C03662=1146.416,331.049,-77.493,-176.659,8.929,148.817
C03663=1146.420,330.801,-77.460,-176.662,8.926,148.817
C03664=1146.424,330.554,-77.428,-176.665,8.922,148.817
C03665=1146.427,330.305,-77.394,-176.667,8.919,148.817
C03666=1146.431,330.057,-77.361,-176.670,8.914,148.816
C03667=1146.436,329.809,-77.329,-176.672,8.911,148.816
C03668=1146.440,329.561,-77.296,-176.675,8.907,148.816
C03669=1146.444,329.314,-77.262,-176.677,8.904,148.816
C03670=1146.448,329.066,-77.229,-176.680,8.900,148.815
C03671=1146.452,328.818,-77.196,-176.682,8.896,148.815
C03672=1146.456,328.571,-77.163,-176.685,8.892,148.815
C03673=1146.460,328.323,-77.130,-176.687,8.889,148.815
C03674=1146.464,328.075,-77.098,-176.690,8.886,148.814
C03675=1146.468,327.827,-77.065,-176.693,8.881,148.814
C03676=1146.472,327.579,-77.032,-176.695,8.878,148.814
C03677=1146.477,327.331,-76.998,-176.698,8.874,148.814
C03678=1146.480,327.083,-76.967,-176.700,8.871,148.814
C03679=1146.484,326.836,-76.933,-176.703,8.867,148.813
C03680=1146.489,326.589,-76.901,-176.705,8.863,148.813
C03681=1146.494,326.340,-76.868,-176.708,8.859,148.813
C03682=1146.497,326.093,-76.836,-176.711,8.856,148.813
C03683=1146.501,325.845,-76.802,-176.713,8.853,148.813
C03684=1146.506,325.597,-76.770,-176.716,8.849,148.812
C03685=1146.509,325.349,-76.737,-176.718,8.846,148.812
C03686=1146.513,325.102,-76.704,-176.721,8.841,148.812
C03687=1146.518,324.853,-76.672,-176.724,8.838,148.812
C03688=1146.522,324.606,-76.639,-176.726,8.834,148.811
C03689=1146.525,324.357,-76.607,-176.729,8.831,148.811
C03690=1146.530,324.110,-76.574,-176.731,8.828,148.811
C03691=1146.534,323.862,-76.541,-176.734,8.823,148.811
C03692=1146.537,323.614,-76.509,-176.736,8.820,148.811
C03693=1146.542,323.366,-76.476,-176.739,8.816,148.810
C03694=1146.546,323.119,-76.444,-176.742,8.813,148.810
C03695=1146.550,322.871,-76.411,-176.745,8.809,148.810
C03696=1146.554,322.623,-76.378,-176.747,8.805,148.810
C03697=1146.558,322.375,-76.346,-176.749,8.802,148.810
C03698=1146.562,322.127,-76.313,-176.752,8.798,148.809
C03699=1146.566,321.880,-76.281,-176.754,8.795,148.809
C03700=1146.570,321.631,-76.248,-176.757,8.791,148.809
C03701=1146.575,321.383,-76.216,-176.760,8.788,148.809
C03702=1146.579,321.136,-76.184,-176.762,8.784,148.809
C03703=1146.583,320.888,-76.151,-176.765,8.780,148.808
C03704=1146.587,320.640,-76.120,-176.767,8.777,148.808
C03705=1146.591,320.392,-76.086,-176.770,8.773,148.808
C03706=1146.595,320.144,-76.055,-176.773,8.770,148.808
C03707=1146.599,319.896,-76.022,-176.775,8.767,148.808
C03708=1146.603,319.649,-75.990,-176.778,8.763,148.808
C03709=1146.607,319.401,-75.957,-176.780,8.759,148.807
C03710=1146.611,319.153,-75.926,-176.783,8.755,148.807
C03711=1146.615,318.905,-75.892,-176.786,8.752,148.807
C03712=1146.619,318.657,-75.861,-176.788,8.749,148.807
C03713=1146.624,318.409,-75.829,-176.791,8.745,148.807
C03714=1146.628,318.161,-75.797,-176.793,8.741,148.806
C03715=1146.631,317.914,-75.764,-176.796,8.737,148.806
C03716=1146.636,317.665,-75.732,-176.799,8.734,148.806
C03717=1146.640,317.418,-75.700,-176.801,8.731,148.806
C03718=1146.644,317.170,-75.668,-176.804,8.727,148.806
C03719=1146.648,316.922,-75.636,-176.807,8.724,148.806
C03720=1146.653,316.673,-75.604,-176.809,8.720,148.805
C03721=1146.657,316.426,-75.572,-176.812,8.716,148.805
C03722=1146.660,316.179,-75.539,-176.814,8.713,148.805
C03723=1146.665,315.930,-75.507,-176.817,8.709,148.805
C03724=1146.668,315.682,-75.475,-176.819,8.706,148.805
C03725=1146.673,315.435,-75.444,-176.822,8.702,148.804
C03726=1146.677,315.186,-75.411,-176.825,8.699,148.804
C03727=1146.681,314.938,-75.379,-176.827,8.695,148.804
C03728=1146.685,314.691,-75.348,-176.830,8.692,148.804
C03729=1146.690,314.443,-75.315,-176.833,8.688,148.804
C03730=1146.693,314.195,-75.284,-176.835,8.685,148.804
C03731=1146.697,313.947,-75.252,-176.837,8.681,148.803
C03732=1146.703,313.670,-75.216,-176.841,8.678,148.803
C03733=1146.707,313.392,-75.180,-176.844,8.674,148.803
C03734=1146.712,313.114,-75.145,-176.846,8.670,148.803
C03735=1146.717,312.836,-75.109,-176.849,8.665,148.803
C03736=1146.720,312.588,-75.077,-176.852,8.662,148.802
C03737=1146.724,312.340,-75.046,-176.855,8.658,148.802
C03738=1146.728,312.093,-75.014,-176.857,8.655,148.802
C03739=1146.733,311.844,-74.982,-176.860,8.652,148.802
C03740=1146.737,311.597,-74.950,-176.863,8.648,148.802
C03741=1146.741,311.348,-74.919,-176.865,8.645,148.802
C03742=1146.745,311.100,-74.887,-176.868,8.642,148.802
C03743=1146.749,310.853,-74.856,-176.871,8.638,148.801
C03744=1146.754,310.605,-74.823,-176.873,8.634,148.801
C03745=1146.757,310.357,-74.791,-176.875,8.631,148.801
C03746=1146.762,310.109,-74.761,-176.878,8.627,148.801
C03747=1146.766,309.861,-74.729,-176.881,8.624,148.801
C03748=1146.770,309.613,-74.697,-176.883,8.621,148.801
C03749=1146.774,309.365,-74.666,-176.886,8.617,148.800
C03750=1146.778,309.117,-74.635,-176.888,8.613,148.800
C03751=1146.783,308.869,-74.602,-176.891,8.610,148.800
C03752=1146.786,308.621,-74.570,-176.894,8.606,148.800
C03753=1146.791,308.373,-74.540,-176.896,8.603,148.800
C03754=1146.795,308.125,-74.508,-176.899,8.600,148.800
C03755=1146.799,307.877,-74.477,-176.902,8.596,148.800
C03756=1146.803,307.629,-74.445,-176.905,8.593,148.800
C03757=1146.807,307.381,-74.414,-176.907,8.589,148.799
C03758=1146.811,307.133,-74.383,-176.910,8.585,148.799
C03759=1146.816,306.885,-74.351,-176.913,8.582,148.799
C03760=1146.820,306.637,-74.320,-176.915,8.579,148.799
C03761=1146.824,306.389,-74.289,-176.918,8.575,148.799
C03762=1146.828,306.141,-74.257,-176.920,8.572,148.799
C03763=1146.832,305.893,-74.226,-176.923,8.569,148.799
C03764=1146.836,305.645,-74.195,-176.925,8.566,148.798
C03765=1146.841,305.397,-74.163,-176.928,8.562,148.798
C03766=1146.845,305.149,-74.132,-176.931,8.559,148.798
C03767=1146.849,304.901,-74.101,-176.933,8.555,148.798
C03768=1146.853,304.653,-74.070,-176.936,8.551,148.798
C03769=1146.857,304.405,-74.038,-176.938,8.548,148.798
C03770=1146.861,304.157,-74.007,-176.941,8.545,148.798
C03771=1146.866,303.909,-73.976,-176.944,8.541,148.798
C03772=1146.870,303.662,-73.945,-176.946,8.538,148.797
C03773=1146.874,303.413,-73.914,-176.949,8.535,148.797
C03774=1146.878,303.166,-73.882,-176.952,8.531,148.797
C03775=1146.883,302.917,-73.851,-176.954,8.527,148.797
C03776=1146.887,302.669,-73.820,-176.957,8.524,148.797
C03777=1146.891,302.420,-73.789,-176.960,8.521,148.797
C03778=1146.895,302.173,-73.758,-176.962,8.517,148.797
C03779=1146.900,301.925,-73.727,-176.965,8.514,148.797
C03780=1146.903,301.677,-73.696,-176.968,8.511,148.796
C03781=1146.908,301.429,-73.665,-176.970,8.508,148.796
C03782=1146.912,301.181,-73.634,-176.973,8.504,148.796
C03783=1146.916,300.933,-73.603,-176.976,8.501,148.796
C03784=1146.921,300.685,-73.572,-176.978,8.497,148.796
C03785=1146.925,300.436,-73.541,-176.981,8.494,148.796
C03786=1146.928,300.189,-73.510,-176.984,8.490,148.796
C03787=1146.932,299.940,-73.479,-176.986,8.487,148.796
C03788=1146.937,299.692,-73.448,-176.989,8.484,148.796
C03789=1146.942,299.444,-73.418,-176.992,8.480,148.795
C03790=1146.946,299.196,-73.386,-176.994,8.477,148.795
C03791=1146.950,298.948,-73.356,-176.997,8.474,148.795
C03792=1146.954,298.700,-73.325,-176.999,8.471,148.795
C03793=1146.958,298.451,-73.294,-177.002,8.467,148.795
C03794=1146.963,298.204,-73.263,-177.005,8.464,148.795
C03795=1146.966,297.957,-73.233,-177.007,8.461,148.795
C03796=1146.970,297.708,-73.202,-177.010,8.457,148.795
C03797=1146.975,297.460,-73.171,-177.013,8.454,148.795
C03798=1146.979,297.212,-73.141,-177.015,8.450,148.795
C03799=1146.983,296.964,-73.109,-177.018,8.447,148.794
C03800=1146.988,296.716,-73.079,-177.021,8.444,148.794
C03801=1146.991,296.468,-73.049,-177.023,8.440,148.794
C03802=1146.996,296.220,-73.018,-177.026,8.437,148.794
C03803=1147.000,295.971,-72.987,-177.029,8.434,148.794
C03804=1147.004,295.723,-72.957,-177.031,8.431,148.794
C03805=1147.009,295.475,-72.926,-177.034,8.427,148.794
C03806=1147.013,295.226,-72.895,-177.037,8.423,148.794
C03807=1147.017,294.979,-72.865,-177.039,8.421,148.794
C03808=1147.021,294.731,-72.834,-177.042,8.417,148.794
C03809=1147.025,294.483,-72.804,-177.044,8.414,148.794
C03810=1147.029,294.235,-72.773,-177.047,8.410,148.793
C03811=1147.034,293.987,-72.742,-177.050,8.407,148.793
C03812=1147.038,293.738,-72.713,-177.052,8.404,148.793
C03813=1147.043,293.490,-72.682,-177.055,8.401,148.793
C03814=1147.046,293.242,-72.652,-177.058,8.397,148.793
C03815=1147.051,292.994,-72.621,-177.060,8.394,148.793
C03816=1147.054,292.746,-72.591,-177.063,8.391,148.793
C03817=1147.059,292.498,-72.561,-177.066,8.388,148.793
C03818=1147.063,292.250,-72.530,-177.068,8.385,148.793
C03819=1147.067,292.002,-72.499,-177.071,8.381,148.793
C03820=1147.071,291.753,-72.470,-177.074,8.378,148.793
C03821=1147.076,291.505,-72.439,-177.076,8.374,148.792
C03822=1147.080,291.258,-72.409,-177.079,8.371,148.793
C03823=1147.084,291.010,-72.378,-177.082,8.367,148.792
C03824=1147.088,290.761,-72.348,-177.085,8.364,148.792
C03825=1147.093,290.513,-72.318,-177.087,8.361,148.792
C03826=1147.097,290.265,-72.288,-177.090,8.358,148.792
C03827=1147.101,290.017,-72.258,-177.092,8.355,148.792
C03828=1147.105,289.769,-72.227,-177.096,8.351,148.792
C03829=1147.110,289.521,-72.198,-177.098,8.348,148.792
C03830=1147.114,289.273,-72.167,-177.101,8.345,148.792
C03831=1147.118,289.024,-72.137,-177.103,8.342,148.792
C03832=1147.122,288.776,-72.106,-177.106,8.339,148.792
C03833=1147.127,288.528,-72.077,-177.109,8.335,148.792
C03834=1147.130,288.280,-72.047,-177.112,8.332,148.792
C03835=1147.135,288.031,-72.017,-177.114,8.329,148.792
C03836=1147.140,287.757,-71.983,-177.117,8.325,148.791
C03837=1147.144,287.481,-71.950,-177.120,8.322,148.792
C03838=1147.149,287.206,-71.917,-177.123,8.318,148.791
C03839=1147.154,286.930,-71.883,-177.126,8.315,148.791
C03840=1147.158,286.682,-71.853,-177.129,8.311,148.791
C03841=1147.162,286.434,-71.823,-177.131,8.308,148.791
C03842=1147.167,286.185,-71.793,-177.134,8.305,148.791
C03843=1147.171,285.937,-71.764,-177.136,8.301,148.791
C03844=1147.175,285.689,-71.734,-177.139,8.299,148.791
C03845=1147.179,285.441,-71.704,-177.142,8.294,148.791
C03846=1147.184,285.193,-71.674,-177.145,8.292,148.791
C03847=1147.188,284.945,-71.644,-177.148,8.289,148.791
C03848=1147.192,284.697,-71.614,-177.150,8.285,148.791
C03849=1147.196,284.448,-71.585,-177.153,8.282,148.791
C03850=1147.201,284.200,-71.554,-177.155,8.279,148.791
C03851=1147.205,283.952,-71.525,-177.158,8.275,148.791
C03852=1147.209,283.704,-71.495,-177.161,8.272,148.791
C03853=1147.213,283.456,-71.466,-177.164,8.269,148.791
C03854=1147.217,283.208,-71.436,-177.166,8.266,148.791
C03855=1147.222,282.959,-71.406,-177.169,8.263,148.790
C03856=1147.226,282.711,-71.376,-177.171,8.260,148.791
C03857=1147.230,282.463,-71.347,-177.175,8.256,148.791
C03858=1147.235,282.215,-71.317,-177.177,8.253,148.790
C03859=1147.239,281.966,-71.288,-177.180,8.250,148.790
C03860=1147.243,281.719,-71.258,-177.182,8.247,148.790
C03861=1147.248,281.470,-71.228,-177.185,8.244,148.790
C03862=1147.252,281.222,-71.198,-177.188,8.241,148.790
C03863=1147.256,280.974,-71.169,-177.190,8.238,148.790
C03864=1147.260,280.725,-71.139,-177.193,8.234,148.790
C03865=1147.264,280.477,-71.110,-177.196,8.231,148.790
C03866=1147.268,280.229,-71.080,-177.199,8.228,148.790
C03867=1147.273,279.981,-71.051,-177.201,8.225,148.790
C03868=1147.277,279.732,-71.021,-177.204,8.222,148.790
C03869=1147.281,279.484,-70.992,-177.206,8.219,148.790
C03870=1147.286,279.236,-70.963,-177.209,8.216,148.790
C03871=1147.290,278.988,-70.933,-177.213,8.212,148.790
C03872=1147.294,278.740,-70.904,-177.215,8.209,148.790
C03873=1147.298,278.492,-70.874,-177.218,8.206,148.790
C03874=1147.303,278.243,-70.845,-177.220,8.203,148.790
C03875=1147.307,277.995,-70.816,-177.223,8.199,148.790
C03876=1147.311,277.747,-70.786,-177.226,8.197,148.790
C03877=1147.315,277.499,-70.757,-177.228,8.194,148.790
C03878=1147.319,277.250,-70.727,-177.231,8.190,148.790
C03879=1147.323,277.002,-70.698,-177.234,8.187,148.790
C03880=1147.328,276.754,-70.669,-177.237,8.184,148.790
C03881=1147.333,276.506,-70.640,-177.239,8.180,148.790
C03882=1147.337,276.257,-70.610,-177.242,8.177,148.790
C03883=1147.341,276.009,-70.581,-177.245,8.174,148.790
C03884=1147.345,275.761,-70.552,-177.247,8.171,148.790
C03885=1147.349,275.513,-70.522,-177.250,8.168,148.790
C03886=1147.354,275.264,-70.494,-177.253,8.165,148.790
C03887=1147.359,275.016,-70.464,-177.255,8.162,148.790
C03888=1147.363,274.768,-70.435,-177.258,8.158,148.790
C03889=1147.367,274.520,-70.405,-177.261,8.155,148.790
C03890=1147.371,274.271,-70.377,-177.264,8.152,148.790
C03891=1147.375,274.023,-70.348,-177.266,8.149,148.790
C03892=1147.380,273.775,-70.319,-177.269,8.146,148.790
C03893=1147.384,273.526,-70.290,-177.272,8.143,148.790
C03894=1147.388,273.278,-70.261,-177.274,8.140,148.790
C03895=1147.393,273.030,-70.231,-177.277,8.137,148.790
C03896=1147.397,272.782,-70.203,-177.280,8.134,148.790
C03897=1147.401,272.534,-70.174,-177.282,8.131,148.790
C03898=1147.405,272.285,-70.144,-177.286,8.127,148.790
C03899=1147.410,272.036,-70.116,-177.288,8.124,148.789
C03900=1147.414,271.788,-70.086,-177.291,8.121,148.790
C03901=1147.418,271.540,-70.058,-177.294,8.118,148.790
C03902=1147.423,271.292,-70.029,-177.296,8.115,148.790
C03903=1147.427,271.043,-70.000,-177.299,8.112,148.789
C03904=1147.431,270.795,-69.971,-177.302,8.109,148.790
C03905=1147.435,270.548,-69.942,-177.304,8.106,148.790
C03906=1147.440,270.299,-69.914,-177.307,8.103,148.790
C03907=1147.444,270.050,-69.885,-177.309,8.100,148.789
C03908=1147.449,269.802,-69.856,-177.312,8.097,148.790
C03909=1147.453,269.554,-69.828,-177.315,8.094,148.790
C03910=1147.457,269.305,-69.798,-177.318,8.090,148.790
C03911=1147.462,269.057,-69.770,-177.321,8.087,148.789
C03912=1147.465,268.809,-69.741,-177.323,8.084,148.790
C03913=1147.470,268.560,-69.712,-177.326,8.081,148.790
C03914=1147.475,268.313,-69.683,-177.329,8.078,148.790
C03915=1147.478,268.064,-69.655,-177.332,8.075,148.790
C03916=1147.483,267.815,-69.626,-177.334,8.072,148.790
C03917=1147.488,267.568,-69.597,-177.337,8.069,148.790
C03918=1147.491,267.319,-69.569,-177.340,8.066,148.790
C03919=1147.496,267.070,-69.540,-177.342,8.063,148.790
C03920=1147.500,266.823,-69.512,-177.345,8.060,148.790
C03921=1147.505,266.574,-69.483,-177.348,8.057,148.790
C03922=1147.509,266.325,-69.454,-177.350,8.054,148.790
C03923=1147.513,266.077,-69.426,-177.353,8.051,148.790
C03924=1147.518,265.829,-69.397,-177.356,8.048,148.790
C03925=1147.521,265.581,-69.369,-177.359,8.045,148.790
C03926=1147.526,265.332,-69.340,-177.361,8.043,148.790
C03927=1147.531,265.083,-69.312,-177.364,8.038,148.790
C03928=1147.535,264.836,-69.283,-177.367,8.036,148.790
C03929=1147.539,264.587,-69.255,-177.370,8.033,148.790
C03930=1147.543,264.339,-69.226,-177.373,8.030,148.790
C03931=1147.548,264.091,-69.198,-177.375,8.027,148.790
C03932=1147.552,263.842,-69.170,-177.378,8.024,148.790
C03933=1147.557,263.594,-69.141,-177.381,8.021,148.790
C03934=1147.561,263.345,-69.113,-177.383,8.018,148.790
C03935=1147.566,263.098,-69.084,-177.386,8.015,148.790
C03936=1147.569,262.849,-69.056,-177.389,8.012,148.790
C03937=1147.574,262.601,-69.028,-177.392,8.009,148.790
C03938=1147.578,262.352,-69.000,-177.394,8.006,148.790
C03939=1147.582,262.104,-68.971,-177.397,8.003,148.790
C03940=1147.587,261.830,-68.940,-177.400,8.000,148.790
C03941=1147.592,261.557,-68.910,-177.403,7.996,148.790
C03942=1147.597,261.283,-68.879,-177.406,7.993,148.790
C03943=1147.602,261.010,-68.847,-177.409,7.989,148.790
C03944=1147.606,260.762,-68.819,-177.412,7.986,148.790
C03945=1147.611,260.514,-68.790,-177.415,7.983,148.790
C03946=1147.614,260.265,-68.762,-177.417,7.980,148.790
C03947=1147.619,260.017,-68.735,-177.420,7.977,148.790
C03948=1147.623,259.768,-68.706,-177.423,7.975,148.790
C03949=1147.628,259.520,-68.679,-177.426,7.972,148.791
C03950=1147.632,259.271,-68.650,-177.429,7.969,148.791
C03951=1147.637,259.023,-68.622,-177.431,7.965,148.790
C03952=1147.640,258.774,-68.594,-177.434,7.963,148.791
C03953=1147.645,258.527,-68.566,-177.436,7.960,148.791
C03954=1147.650,258.278,-68.538,-177.439,7.957,148.791
C03955=1147.654,258.029,-68.510,-177.442,7.954,148.791
C03956=1147.658,257.781,-68.483,-177.445,7.951,148.791
C03957=1147.662,257.533,-68.454,-177.448,7.948,148.791
C03958=1147.667,257.285,-68.426,-177.450,7.945,148.791
C03959=1147.671,257.036,-68.398,-177.453,7.942,148.791
C03960=1147.676,256.788,-68.371,-177.456,7.939,148.791
C03961=1147.679,256.539,-68.343,-177.459,7.936,148.791
C03962=1147.684,256.291,-68.314,-177.461,7.933,148.791
C03963=1147.689,256.043,-68.287,-177.464,7.930,148.791
C03964=1147.693,255.794,-68.259,-177.467,7.927,148.791
C03965=1147.697,255.546,-68.231,-177.469,7.924,148.791
C03966=1147.702,255.297,-68.203,-177.472,7.921,148.791
C03967=1147.706,255.048,-68.176,-177.475,7.918,148.791
C03968=1147.711,254.801,-68.148,-177.478,7.915,148.791
C03969=1147.714,254.552,-68.120,-177.481,7.912,148.791
C03970=1147.719,254.303,-68.093,-177.483,7.909,148.791
C03971=1147.723,254.056,-68.065,-177.486,7.906,148.792
C03972=1147.728,253.806,-68.037,-177.489,7.904,148.792
C03973=1147.733,253.558,-68.009,-177.492,7.901,148.792
C03974=1147.737,253.310,-67.981,-177.494,7.899,148.792
C03975=1147.741,253.061,-67.954,-177.497,7.896,148.792
C03976=1147.745,252.813,-67.926,-177.499,7.893,148.792
C03977=1147.750,252.565,-67.899,-177.502,7.890,148.792
C03978=1147.754,252.316,-67.871,-177.505,7.887,148.792
C03979=1147.758,252.068,-67.844,-177.508,7.884,148.792
C03980=1147.763,251.820,-67.816,-177.511,7.881,148.792
C03981=1147.767,251.571,-67.789,-177.513,7.878,148.792
C03982=1147.771,251.323,-67.761,-177.516,7.875,148.792
C03983=1147.776,251.074,-67.733,-177.519,7.872,148.792
C03984=1147.780,250.825,-67.705,-177.521,7.869,148.792
C03985=1147.785,250.577,-67.678,-177.524,7.866,148.792
C03986=1147.790,250.328,-67.651,-177.527,7.863,148.792
C03987=1147.793,250.080,-67.623,-177.530,7.860,148.792
C03988=1147.798,249.831,-67.596,-177.532,7.857,148.793
C03989=1147.803,249.583,-67.569,-177.535,7.854,148.793
C03990=1147.807,249.335,-67.541,-177.538,7.851,148.793
C03991=1147.811,249.086,-67.513,-177.541,7.848,148.793
C03992=1147.815,248.838,-67.486,-177.544,7.845,148.793
C03993=1147.820,248.589,-67.459,-177.546,7.843,148.793
C03994=1147.824,248.341,-67.432,-177.549,7.840,148.793
C03995=1147.828,248.092,-67.405,-177.551,7.837,148.793
C03996=1147.832,247.844,-67.377,-177.554,7.835,148.793
C03997=1147.837,247.596,-67.350,-177.557,7.832,148.793
C03998=1147.842,247.347,-67.323,-177.560,7.829,148.794
C03999=1147.846,247.099,-67.296,-177.563,7.826,148.794
C04000=1147.850,246.850,-67.268,-177.566,7.823,148.794
C04001=1147.855,246.602,-67.241,-177.568,7.820,148.794
C04002=1147.859,246.353,-67.213,-177.571,7.817,148.794
C04003=1147.864,246.105,-67.186,-177.574,7.814,148.794
C04004=1147.869,245.856,-67.159,-177.577,7.811,148.794
C04005=1147.872,245.608,-67.132,-177.580,7.809,148.794
C04006=1147.876,245.359,-67.105,-177.582,7.806,148.794
C04007=1147.881,245.111,-67.078,-177.585,7.803,148.794
C04008=1147.886,244.862,-67.051,-177.588,7.800,148.794
C04009=1147.890,244.614,-67.024,-177.590,7.798,148.794
C04010=1147.895,244.365,-66.996,-177.593,7.795,148.794
C04011=1147.898,244.116,-66.970,-177.596,7.792,148.794
C04012=1147.903,243.868,-66.943,-177.599,7.789,148.795
C04013=1147.908,243.619,-66.916,-177.601,7.786,148.795
C04014=1147.912,243.371,-66.888,-177.604,7.783,148.795
C04015=1147.916,243.123,-66.862,-177.607,7.780,148.795
C04016=1147.921,242.874,-66.835,-177.610,7.777,148.795
C04017=1147.926,242.626,-66.808,-177.613,7.774,148.795
C04018=1147.930,242.377,-66.781,-177.615,7.771,148.795
C04019=1147.933,242.128,-66.754,-177.617,7.769,148.795
C04020=1147.938,241.880,-66.727,-177.621,7.767,148.795
C04021=1147.943,241.631,-66.700,-177.624,7.764,148.795
C04022=1147.947,241.383,-66.673,-177.626,7.761,148.796
C04023=1147.951,241.135,-66.646,-177.629,7.758,148.796
C04024=1147.956,240.886,-66.619,-177.632,7.755,148.796
C04025=1147.961,240.638,-66.592,-177.635,7.752,148.796
C04026=1147.965,240.390,-66.566,-177.637,7.749,148.796
C04027=1147.970,240.140,-66.539,-177.640,7.746,148.796
C04028=1147.974,239.892,-66.512,-177.642,7.744,148.796
C04029=1147.978,239.644,-66.486,-177.645,7.741,148.796
C04030=1147.983,239.395,-66.459,-177.648,7.738,148.796
C04031=1147.987,239.147,-66.432,-177.651,7.736,148.797
C04032=1147.991,238.899,-66.405,-177.654,7.733,148.797
C04033=1147.996,238.649,-66.379,-177.657,7.730,148.797
C04034=1148.000,238.401,-66.352,-177.660,7.727,148.797
C04035=1148.004,238.152,-66.325,-177.662,7.724,148.797
C04036=1148.009,237.904,-66.298,-177.665,7.722,148.797
C04037=1148.013,237.655,-66.272,-177.667,7.719,148.797
C04038=1148.018,237.406,-66.245,-177.670,7.716,148.797
C04039=1148.022,237.158,-66.219,-177.673,7.713,148.797
C04040=1148.027,236.909,-66.192,-177.676,7.710,148.797
C04041=1148.031,236.661,-66.166,-177.679,7.708,148.798
C04042=1148.035,236.412,-66.139,-177.682,7.705,148.798
C04043=1148.040,236.164,-66.113,-177.684,7.702,148.798
C04044=1148.045,235.892,-66.084,-177.687,7.699,148.798
C04045=1148.050,235.620,-66.054,-177.690,7.696,148.798
C04046=1148.054,235.348,-66.026,-177.693,7.693,148.798
C04047=1148.060,235.077,-65.997,-177.696,7.690,148.798
C04048=1148.064,234.829,-65.971,-177.699,7.687,148.798
C04049=1148.068,234.579,-65.944,-177.702,7.684,148.798
C04050=1148.072,234.331,-65.918,-177.705,7.682,148.798
C04051=1148.077,234.082,-65.891,-177.707,7.679,148.799
C04052=1148.081,233.834,-65.865,-177.710,7.677,148.799
C04053=1148.086,233.585,-65.839,-177.713,7.674,148.799
C04054=1148.090,233.337,-65.812,-177.716,7.671,148.799
C04055=1148.095,233.088,-65.786,-177.718,7.668,148.799
C04056=1148.099,232.839,-65.759,-177.721,7.665,148.799
C04057=1148.104,232.591,-65.734,-177.724,7.662,148.799
C04058=1148.109,232.343,-65.707,-177.727,7.660,148.800
C04059=1148.113,232.094,-65.681,-177.729,7.658,148.800
C04060=1148.118,231.845,-65.655,-177.732,7.655,148.800
C04061=1148.122,231.597,-65.628,-177.735,7.652,148.800
C04062=1148.126,231.348,-65.603,-177.738,7.649,148.800
C04063=1148.131,231.099,-65.575,-177.741,7.646,148.800
C04064=1148.135,230.851,-65.550,-177.743,7.644,148.800
C04065=1148.140,230.602,-65.524,-177.746,7.641,148.800
C04066=1148.144,230.354,-65.497,-177.749,7.638,148.801
C04067=1148.148,230.105,-65.471,-177.752,7.635,148.801
C04068=1148.153,229.856,-65.446,-177.754,7.632,148.801
C04069=1148.157,229.608,-65.419,-177.757,7.630,148.801
C04070=1148.162,229.359,-65.393,-177.760,7.628,148.801
C04071=1148.166,229.110,-65.367,-177.763,7.625,148.801
C04072=1148.171,228.862,-65.342,-177.766,7.622,148.801
C04073=1148.175,228.614,-65.315,-177.768,7.619,148.801
C04074=1148.179,228.365,-65.289,-177.771,7.617,148.802
C04075=1148.184,228.116,-65.263,-177.774,7.614,148.802
C04076=1148.188,227.867,-65.237,-177.777,7.611,148.802
C04077=1148.193,227.619,-65.211,-177.779,7.608,148.802
C04078=1148.197,227.371,-65.185,-177.782,7.605,148.802
C04079=1148.202,227.122,-65.159,-177.785,7.604,148.802
C04080=1148.206,226.873,-65.134,-177.788,7.601,148.803
C04081=1148.211,226.625,-65.108,-177.790,7.598,148.803
C04082=1148.216,226.376,-65.082,-177.793,7.595,148.803
C04083=1148.220,226.127,-65.056,-177.796,7.592,148.803
C04084=1148.224,225.879,-65.030,-177.799,7.590,148.803
C04085=1148.228,225.630,-65.004,-177.801,7.587,148.803
C04086=1148.233,225.382,-64.978,-177.804,7.584,148.803
C04087=1148.237,225.133,-64.953,-177.807,7.582,148.803
C04088=1148.242,224.884,-64.926,-177.810,7.580,148.804
C04089=1148.247,224.636,-64.901,-177.812,7.577,148.804
C04090=1148.251,224.387,-64.875,-177.815,7.574,148.804
C04091=1148.255,224.138,-64.849,-177.818,7.571,148.804
C04092=1148.260,223.890,-64.824,-177.820,7.569,148.804
C04093=1148.264,223.641,-64.798,-177.824,7.566,148.804
C04094=1148.269,223.393,-64.773,-177.826,7.563,148.804
C04095=1148.273,223.144,-64.747,-177.829,7.560,148.805
C04096=1148.278,222.896,-64.721,-177.832,7.558,148.805
C04097=1148.282,222.647,-64.696,-177.835,7.556,148.805
C04098=1148.286,222.398,-64.670,-177.837,7.553,148.805
C04099=1148.292,222.149,-64.645,-177.840,7.550,148.805
C04100=1148.296,221.900,-64.619,-177.843,7.547,148.805
C04101=1148.300,221.651,-64.593,-177.846,7.545,148.806
C04102=1148.305,221.403,-64.568,-177.848,7.542,148.806
C04103=1148.309,221.155,-64.542,-177.851,7.539,148.806
C04104=1148.314,220.906,-64.516,-177.854,7.538,148.806
C04105=1148.319,220.658,-64.491,-177.857,7.535,148.806
C04106=1148.323,220.408,-64.466,-177.859,7.532,148.806
C04107=1148.327,220.159,-64.440,-177.862,7.529,148.806
C04108=1148.331,219.912,-64.415,-177.865,7.527,148.807
C04109=1148.336,219.663,-64.390,-177.868,7.524,148.807
C04110=1148.340,219.414,-64.364,-177.871,7.521,148.807
C04111=1148.345,219.165,-64.339,-177.874,7.519,148.807
C04112=1148.349,218.916,-64.313,-177.876,7.517,148.807
C04113=1148.354,218.668,-64.288,-177.879,7.514,148.807
C04114=1148.358,218.420,-64.262,-177.882,7.511,148.808
C04115=1148.363,218.170,-64.237,-177.885,7.508,148.808
C04116=1148.368,217.922,-64.212,-177.887,7.506,148.808
C04117=1148.372,217.673,-64.186,-177.890,7.503,148.808
C04118=1148.377,217.424,-64.161,-177.893,7.501,148.808
C04119=1148.380,217.176,-64.136,-177.895,7.499,148.809
C04120=1148.385,216.928,-64.111,-177.898,7.496,148.809
C04121=1148.390,216.678,-64.086,-177.901,7.493,148.809
C04122=1148.394,216.430,-64.060,-177.904,7.491,148.809
C04123=1148.399,216.181,-64.035,-177.906,7.488,148.809
C04124=1148.403,215.932,-64.010,-177.910,7.485,148.809
C04125=1148.407,215.684,-63.985,-177.912,7.483,148.810
C04126=1148.412,215.435,-63.960,-177.915,7.480,148.810
C04127=1148.417,215.187,-63.934,-177.917,7.477,148.810
C04128=1148.421,214.937,-63.909,-177.921,7.475,148.810
C04129=1148.426,214.689,-63.884,-177.923,7.473,148.810
C04130=1148.430,214.440,-63.860,-177.926,7.470,148.810
C04131=1148.435,214.192,-63.834,-177.929,7.467,148.811
C04132=1148.439,213.943,-63.809,-177.931,7.465,148.811
C04133=1148.444,213.695,-63.784,-177.934,7.462,148.811
C04134=1148.448,213.445,-63.759,-177.937,7.460,148.811
C04135=1148.453,213.197,-63.734,-177.939,7.458,148.811
C04136=1148.457,212.948,-63.709,-177.943,7.455,148.812
C04137=1148.462,212.699,-63.684,-177.946,7.452,148.812
C04138=1148.466,212.451,-63.659,-177.948,7.450,148.812
C04139=1148.471,212.202,-63.634,-177.951,7.447,148.812
C04140=1148.475,211.953,-63.609,-177.954,7.445,148.812
C04141=1148.480,211.705,-63.585,-177.956,7.442,148.812
C04142=1148.484,211.455,-63.560,-177.959,7.440,148.813
C04143=1148.489,211.207,-63.534,-177.962,7.437,148.813
C04144=1148.493,210.959,-63.510,-177.964,7.435,148.813
C04145=1148.498,210.709,-63.485,-177.968,7.432,148.813
C04146=1148.503,210.461,-63.460,-177.970,7.429,148.813
C04147=1148.507,210.212,-63.435,-177.973,7.428,148.814
C04148=1148.512,209.942,-63.409,-177.976,7.425,148.814
C04149=1148.517,209.671,-63.381,-177.979,7.422,148.814
C04150=1148.522,209.401,-63.354,-177.982,7.419,148.814
C04151=1148.527,209.130,-63.327,-177.985,7.417,148.814
C04152=1148.531,208.881,-63.303,-177.988,7.414,148.815
C04153=1148.536,208.632,-63.278,-177.991,7.411,148.815
C04154=1148.541,208.383,-63.253,-177.993,7.409,148.815
C04155=1148.545,208.135,-63.229,-177.996,7.406,148.815
C04156=1148.549,207.886,-63.203,-177.998,7.404,148.815
C04157=1148.554,207.638,-63.179,-178.002,7.401,148.816
C04158=1148.559,207.389,-63.155,-178.004,7.399,148.816
C04159=1148.563,207.140,-63.130,-178.007,7.397,148.816
C04160=1148.568,206.891,-63.106,-178.010,7.394,148.816
C04161=1148.572,206.643,-63.082,-178.013,7.391,148.816
C04162=1148.577,206.393,-63.057,-178.015,7.389,148.817
C04163=1148.581,206.145,-63.032,-178.018,7.386,148.817
C04164=1148.586,205.897,-63.007,-178.021,7.385,148.817
C04165=1148.590,205.648,-62.983,-178.024,7.382,148.817
C04166=1148.595,205.399,-62.958,-178.027,7.379,148.817
C04167=1148.599,205.150,-62.934,-178.029,7.377,148.818
C04168=1148.604,204.901,-62.909,-178.032,7.374,148.818
C04169=1148.608,204.653,-62.885,-178.035,7.372,148.818
C04170=1148.613,204.404,-62.860,-178.037,7.369,148.818
C04171=1148.617,204.155,-62.836,-178.041,7.367,148.818
C04172=1148.622,203.906,-62.811,-178.043,7.365,148.819
C04173=1148.627,203.658,-62.787,-178.046,7.362,148.819
C04174=1148.631,203.409,-62.763,-178.049,7.359,148.819
C04175=1148.636,203.160,-62.738,-178.052,7.358,148.819
C04176=1148.640,202.911,-62.714,-178.055,7.355,148.819
C04177=1148.645,202.662,-62.690,-178.057,7.353,148.820
C04178=1148.650,202.414,-62.666,-178.060,7.350,148.820
C04179=1148.654,202.164,-62.641,-178.063,7.347,148.820
C04180=1148.659,201.916,-62.617,-178.065,7.345,148.820
C04181=1148.663,201.667,-62.593,-178.068,7.342,148.820
C04182=1148.668,201.419,-62.568,-178.071,7.341,148.821
C04183=1148.672,201.170,-62.543,-178.074,7.338,148.821
C04184=1148.677,200.920,-62.520,-178.076,7.336,148.821
C04185=1148.681,200.672,-62.496,-178.079,7.333,148.821
C04186=1148.686,200.424,-62.472,-178.083,7.330,148.822
C04187=1148.690,200.174,-62.447,-178.085,7.328,148.822
C04188=1148.694,199.926,-62.423,-178.088,7.326,148.822
C04189=1148.699,199.677,-62.399,-178.090,7.324,148.822
C04190=1148.704,199.428,-62.375,-178.093,7.321,148.822
C04191=1148.709,199.180,-62.351,-178.096,7.318,148.823
C04192=1148.713,198.930,-62.327,-178.099,7.316,148.823
C04193=1148.717,198.681,-62.303,-178.102,7.314,148.823
C04194=1148.722,198.433,-62.278,-178.104,7.311,148.823
C04195=1148.727,198.184,-62.254,-178.107,7.309,148.824
C04196=1148.731,197.935,-62.231,-178.109,7.307,148.824
C04197=1148.736,197.687,-62.207,-178.113,7.304,148.824
C04198=1148.740,197.438,-62.182,-178.115,7.302,148.824
C04199=1148.745,197.188,-62.158,-178.118,7.300,148.825
C04200=1148.749,196.940,-62.134,-178.121,7.297,148.825
C04201=1148.754,196.691,-62.111,-178.124,7.295,148.825
C04202=1148.759,196.443,-62.087,-178.127,7.292,148.825
C04203=1148.763,196.194,-62.063,-178.129,7.290,148.826
C04204=1148.768,195.945,-62.039,-178.132,7.287,148.826
C04205=1148.773,195.696,-62.015,-178.135,7.286,148.826
C04206=1148.777,195.447,-61.991,-178.138,7.283,148.826
C04207=1148.781,195.198,-61.967,-178.140,7.281,148.826
C04208=1148.786,194.949,-61.944,-178.143,7.278,148.827
C04209=1148.790,194.701,-61.919,-178.146,7.276,148.827
C04210=1148.795,194.452,-61.896,-178.149,7.274,148.827
C04211=1148.799,194.203,-61.872,-178.151,7.272,148.827
C04212=1148.804,193.954,-61.849,-178.154,7.269,148.828
C04213=1148.809,193.706,-61.825,-178.157,7.266,148.828
C04214=1148.814,193.457,-61.801,-178.160,7.264,148.828
C04215=1148.818,193.208,-61.777,-178.163,7.262,148.828
C04216=1148.823,192.959,-61.753,-178.165,7.260,148.829
C04217=1148.828,192.710,-61.730,-178.168,7.257,148.829
C04218=1148.832,192.462,-61.706,-178.171,7.255,148.829
C04219=1148.836,192.212,-61.682,-178.174,7.252,148.829
C04220=1148.841,191.963,-61.659,-178.176,7.250,148.830
C04221=1148.845,191.715,-61.635,-178.180,7.248,148.830
C04222=1148.850,191.466,-61.611,-178.182,7.246,148.830
C04223=1148.855,191.216,-61.588,-178.185,7.243,148.830
C04224=1148.859,190.968,-61.564,-178.187,7.241,148.831
C04225=1148.864,190.719,-61.540,-178.191,7.239,148.831
C04226=1148.869,190.470,-61.517,-178.193,7.237,148.831
C04227=1148.873,190.222,-61.493,-178.196,7.234,148.831
C04228=1148.878,189.973,-61.470,-178.198,7.232,148.831
C04229=1148.882,189.724,-61.446,-178.202,7.229,148.832
C04230=1148.887,189.474,-61.423,-178.204,7.228,148.832
C04231=1148.891,189.226,-61.399,-178.207,7.225,148.832
C04232=1148.896,188.977,-61.376,-178.210,7.223,148.833
C04233=1148.901,188.729,-61.353,-178.213,7.220,148.833
C04234=1148.905,188.480,-61.330,-178.215,7.218,148.833
C04235=1148.910,188.231,-61.306,-178.219,7.216,148.833
C04236=1148.914,187.983,-61.282,-178.221,7.214,148.834
C04237=1148.919,187.734,-61.259,-178.224,7.211,148.834
C04238=1148.924,187.484,-61.236,-178.226,7.209,148.834
C04239=1148.929,187.235,-61.212,-178.230,7.206,148.834
C04240=1148.933,186.986,-61.189,-178.232,7.204,148.835
C04241=1148.938,186.737,-61.166,-178.234,7.203,148.835
C04242=1148.942,186.489,-61.143,-178.238,7.200,148.835
C04243=1148.947,186.240,-61.119,-178.240,7.198,148.835
C04244=1148.951,185.991,-61.095,-178.243,7.195,148.836
C04245=1148.956,185.742,-61.072,-178.246,7.194,148.836
C04246=1148.960,185.493,-61.049,-178.249,7.191,148.836
C04247=1148.964,185.244,-61.026,-178.251,7.189,148.837
C04248=1148.970,184.996,-61.003,-178.254,7.186,148.837
C04249=1148.974,184.747,-60.980,-178.257,7.184,148.837
C04250=1148.979,184.498,-60.956,-178.260,7.182,148.837
C04251=1148.984,184.249,-60.933,-178.262,7.180,148.838
C04252=1148.988,183.980,-60.908,-178.266,7.177,148.838
C04253=1148.994,183.710,-60.883,-178.269,7.175,148.838
C04254=1148.999,183.440,-60.858,-178.271,7.172,148.838
C04255=1149.004,183.171,-60.833,-178.274,7.170,148.839
C04256=1149.008,182.922,-60.810,-178.277,7.168,148.839
C04257=1149.013,182.673,-60.787,-178.280,7.166,148.839
C04258=1149.018,182.423,-60.764,-178.283,7.164,148.840
C04259=1149.022,182.175,-60.741,-178.286,7.161,148.840
C04260=1149.026,181.926,-60.718,-178.288,7.159,148.840
C04261=1149.031,181.677,-60.694,-178.291,7.156,148.840
C04262=1149.036,181.429,-60.672,-178.294,7.155,148.841
C04263=1149.040,181.180,-60.649,-178.297,7.152,148.841
C04264=1149.045,180.930,-60.626,-178.300,7.150,148.841
C04265=1149.049,180.681,-60.603,-178.302,7.148,148.842
C04266=1149.054,180.432,-60.580,-178.305,7.145,148.842
C04267=1149.059,180.184,-60.557,-178.308,7.144,148.842
C04268=1149.063,179.935,-60.534,-178.311,7.141,148.842
C04269=1149.068,179.686,-60.511,-178.313,7.139,148.843
C04270=1149.072,179.437,-60.489,-178.316,7.137,148.843
C04271=1149.077,179.188,-60.465,-178.319,7.135,148.843
C04272=1149.082,178.939,-60.442,-178.322,7.133,148.843
C04273=1149.086,178.690,-60.420,-178.325,7.130,148.844
C04274=1149.091,178.441,-60.397,-178.328,7.128,148.844
C04275=1149.095,178.192,-60.374,-178.330,7.126,148.844
C04276=1149.101,177.943,-60.352,-178.333,7.124,148.845
C04277=1149.105,177.695,-60.329,-178.336,7.122,148.845
C04278=1149.109,177.446,-60.306,-178.339,7.119,148.845
C04279=1149.114,177.196,-60.283,-178.341,7.117,148.845
C04280=1149.119,176.948,-60.261,-178.344,7.115,148.846
C04281=1149.124,176.699,-60.237,-178.347,7.113,148.846
C04282=1149.128,176.450,-60.215,-178.349,7.111,148.846
C04283=1149.133,176.201,-60.192,-178.353,7.108,148.847
C04284=1149.138,175.952,-60.170,-178.355,7.106,148.847
C04285=1149.142,175.703,-60.147,-178.358,7.104,148.847
C04286=1149.147,175.454,-60.125,-178.361,7.102,148.847
C04287=1149.152,175.205,-60.102,-178.364,7.100,148.848
C04288=1149.156,174.956,-60.079,-178.366,7.097,148.848
C04289=1149.160,174.707,-60.057,-178.369,7.096,148.848
C04290=1149.165,174.459,-60.034,-178.372,7.094,148.849
C04291=1149.170,174.209,-60.012,-178.375,7.091,148.849
C04292=1149.174,173.960,-59.989,-178.377,7.089,148.849
C04293=1149.179,173.712,-59.967,-178.380,7.087,148.850
C04294=1149.184,173.462,-59.944,-178.383,7.085,148.850
C04295=1149.188,173.213,-59.921,-178.385,7.083,148.850
C04296=1149.193,172.965,-59.900,-178.389,7.080,148.850
C04297=1149.198,172.716,-59.876,-178.391,7.079,148.851
C04298=1149.203,172.467,-59.855,-178.394,7.076,148.851
C04299=1149.207,172.218,-59.831,-178.397,7.074,148.851
C04300=1149.212,171.969,-59.809,-178.400,7.072,148.852
C04301=1149.216,171.720,-59.788,-178.402,7.070,148.852
C04302=1149.221,171.471,-59.764,-178.405,7.068,148.852
C04303=1149.225,171.222,-59.742,-178.408,7.066,148.853
C04304=1149.230,170.973,-59.721,-178.411,7.064,148.853
C04305=1149.235,170.724,-59.697,-178.414,7.062,148.853
C04306=1149.240,170.475,-59.676,-178.416,7.059,148.853
C04307=1149.244,170.226,-59.654,-178.419,7.058,148.854
C04308=1149.249,169.978,-59.631,-178.422,7.055,148.854
C04309=1149.254,169.728,-59.608,-178.424,7.053,148.854
C04310=1149.258,169.479,-59.586,-178.427,7.051,148.855
C04311=1149.264,169.230,-59.564,-178.430,7.049,148.855
C04312=1149.267,168.981,-59.541,-178.433,7.047,148.855
C04313=1149.272,168.733,-59.520,-178.435,7.045,148.855
C04314=1149.277,168.483,-59.498,-178.438,7.042,148.856
C04315=1149.282,168.234,-59.475,-178.441,7.041,148.856
C04316=1149.286,167.986,-59.453,-178.444,7.039,148.857
C04317=1149.291,167.737,-59.431,-178.447,7.036,148.857
C04318=1149.295,167.488,-59.409,-178.449,7.034,148.857
C04319=1149.301,167.239,-59.387,-178.452,7.033,148.857
C04320=1149.305,166.989,-59.365,-178.455,7.030,148.858
C04321=1149.310,166.741,-59.343,-178.458,7.028,148.858
C04322=1149.314,166.491,-59.321,-178.460,7.026,148.858
C04323=1149.319,166.243,-59.298,-178.464,7.024,148.859
C04324=1149.324,165.994,-59.276,-178.466,7.022,148.859
C04325=1149.329,165.745,-59.254,-178.469,7.020,148.859
C04326=1149.333,165.496,-59.232,-178.472,7.017,148.860
C04327=1149.338,165.247,-59.210,-178.474,7.016,148.860
C04328=1149.342,164.998,-59.188,-178.477,7.014,148.860
C04329=1149.347,164.749,-59.167,-178.480,7.011,148.861
C04330=1149.351,164.500,-59.145,-178.483,7.010,148.861
C04331=1149.357,164.251,-59.122,-178.485,7.008,148.861
C04332=1149.361,164.002,-59.100,-178.488,7.006,148.862
C04333=1149.366,163.753,-59.079,-178.491,7.003,148.862
C04334=1149.370,163.504,-59.057,-178.494,7.002,148.862
C04335=1149.375,163.255,-59.035,-178.497,7.000,148.863
C04336=1149.379,163.006,-59.013,-178.500,6.997,148.863
C04337=1149.384,162.757,-58.991,-178.502,6.995,148.863
C04338=1149.389,162.508,-58.969,-178.505,6.993,148.864
C04339=1149.393,162.259,-58.947,-178.508,6.992,148.864
C04340=1149.398,162.010,-58.926,-178.511,6.989,148.864
C04341=1149.403,161.761,-58.904,-178.513,6.987,148.864
C04342=1149.408,161.512,-58.883,-178.516,6.985,148.865
C04343=1149.412,161.262,-58.861,-178.519,6.983,148.865
C04344=1149.417,161.014,-58.839,-178.522,6.981,148.866
C04345=1149.422,160.765,-58.817,-178.525,6.979,148.866
C04346=1149.426,160.516,-58.795,-178.527,6.977,148.866
C04347=1149.431,160.267,-58.774,-178.530,6.975,148.866
C04348=1149.435,160.018,-58.751,-178.533,6.973,148.867
C04349=1149.440,159.769,-58.731,-178.536,6.971,148.867
C04350=1149.445,159.520,-58.709,-178.538,6.970,148.868
C04351=1149.450,159.271,-58.687,-178.542,6.967,148.868
C04352=1149.454,159.022,-58.665,-178.544,6.965,148.868
C04353=1149.460,158.773,-58.644,-178.546,6.963,148.868
C04354=1149.464,158.523,-58.622,-178.549,6.961,148.869
C04355=1149.469,158.275,-58.600,-178.552,6.959,148.869
C04356=1149.473,158.006,-58.578,-178.555,6.957,148.870
C04357=1149.479,157.737,-58.554,-178.558,6.955,148.870
C04358=1149.484,157.468,-58.530,-178.561,6.953,148.870
C04359=1149.489,157.198,-58.507,-178.564,6.950,148.871
C04360=1149.494,156.950,-58.486,-178.567,6.949,148.871
C04361=1149.499,156.701,-58.464,-178.570,6.947,148.871
C04362=1149.503,156.451,-58.443,-178.572,6.945,148.872
C04363=1149.508,156.203,-58.421,-178.575,6.942,148.872
C04364=1149.512,155.954,-58.401,-178.578,6.941,148.872
C04365=1149.517,155.704,-58.379,-178.581,6.939,148.873
C04366=1149.522,155.456,-58.357,-178.583,6.937,148.873
C04367=1149.527,155.206,-58.336,-178.587,6.935,148.873
C04368=1149.531,154.957,-58.314,-178.589,6.933,148.874
C04369=1149.536,154.708,-58.293,-178.592,6.931,148.874
C04370=1149.540,154.459,-58.272,-178.594,6.929,148.874
C04371=1149.545,154.211,-58.250,-178.598,6.927,148.875
C04372=1149.550,153.961,-58.229,-178.600,6.925,148.875
C04373=1149.555,153.712,-58.207,-178.603,6.923,148.875
C04374=1149.560,153.463,-58.186,-178.606,6.921,148.876
C04375=1149.564,153.215,-58.165,-178.609,6.920,148.876
C04376=1149.569,152.965,-58.144,-178.612,6.917,148.877
C04377=1149.573,152.716,-58.122,-178.614,6.915,148.877
C04378=1149.579,152.467,-58.101,-178.617,6.913,148.877
C04379=1149.583,152.218,-58.081,-178.619,6.912,148.878
C04380=1149.588,151.969,-58.059,-178.622,6.910,148.878
C04381=1149.592,151.719,-58.038,-178.625,6.907,148.878
C04382=1149.597,151.471,-58.016,-178.628,6.906,148.879
C04383=1149.602,151.222,-57.996,-178.631,6.904,148.879
C04384=1149.607,150.973,-57.974,-178.634,6.902,148.879
C04385=1149.612,150.724,-57.953,-178.636,6.900,148.880
C04386=1149.616,150.474,-57.932,-178.639,6.898,148.880
C04387=1149.621,150.225,-57.911,-178.642,6.896,148.880
C04388=1149.626,149.976,-57.890,-178.645,6.894,148.881
C04389=1149.630,149.727,-57.869,-178.647,6.892,148.881
C04390=1149.635,149.479,-57.848,-178.650,6.891,148.881
C04391=1149.640,149.229,-57.827,-178.653,6.888,148.882
C04392=1149.644,148.980,-57.806,-178.656,6.886,148.882
C04393=1149.649,148.731,-57.784,-178.659,6.885,148.883
C04394=1149.654,148.482,-57.763,-178.661,6.883,148.883
C04395=1149.658,148.233,-57.743,-178.664,6.881,148.883
C04396=1149.664,147.984,-57.722,-178.667,6.880,148.884
C04397=1149.668,147.735,-57.701,-178.670,6.877,148.884
C04398=1149.673,147.486,-57.680,-178.672,6.875,148.884
C04399=1149.678,147.237,-57.659,-178.675,6.873,148.885
C04400=1149.682,146.987,-57.638,-178.678,6.872,148.885
C04401=1149.687,146.738,-57.617,-178.680,6.870,148.885
C04402=1149.691,146.490,-57.596,-178.683,6.868,148.886
C04403=1149.696,146.240,-57.575,-178.686,6.866,148.886
C04404=1149.701,145.991,-57.555,-178.689,6.864,148.887
C04405=1149.706,145.742,-57.534,-178.692,6.862,148.887
C04406=1149.711,145.493,-57.513,-178.695,6.860,148.887
C04407=1149.716,145.244,-57.492,-178.697,6.859,148.888
C04408=1149.721,144.995,-57.472,-178.700,6.857,148.888
C04409=1149.725,144.746,-57.450,-178.703,6.855,148.889
C04410=1149.730,144.497,-57.429,-178.706,6.852,148.889
C04411=1149.734,144.247,-57.409,-178.708,6.851,148.889
C04412=1149.738,143.998,-57.388,-178.711,6.849,148.889
C04413=1149.744,143.749,-57.367,-178.714,6.847,148.890
C04414=1149.748,143.500,-57.347,-178.716,6.845,148.890
C04415=1149.753,143.251,-57.326,-178.719,6.844,148.891
C04416=1149.758,143.002,-57.306,-178.722,6.842,148.891
C04417=1149.763,142.753,-57.285,-178.725,6.840,148.891
C04418=1149.767,142.504,-57.264,-178.728,6.838,148.892
C04419=1149.772,142.254,-57.243,-178.730,6.836,148.892
C04420=1149.777,142.006,-57.223,-178.733,6.834,148.893
C04421=1149.781,141.757,-57.203,-178.736,6.833,148.893
C04422=1149.787,141.507,-57.182,-178.739,6.831,148.893
C04423=1149.791,141.258,-57.161,-178.741,6.829,148.894
C04424=1149.796,141.009,-57.140,-178.744,6.828,148.894
C04425=1149.801,140.760,-57.120,-178.747,6.825,148.894
C04426=1149.805,140.511,-57.100,-178.750,6.823,148.895
C04427=1149.810,140.262,-57.079,-178.753,6.822,148.895
C04428=1149.815,140.012,-57.059,-178.755,6.820,148.896
C04429=1149.819,139.763,-57.039,-178.758,6.818,148.896
C04430=1149.825,139.514,-57.018,-178.761,6.816,148.896
C04431=1149.829,139.265,-56.997,-178.764,6.815,148.897
C04432=1149.833,139.016,-56.977,-178.766,6.813,148.897
C04433=1149.839,138.767,-56.956,-178.769,6.811,148.898
C04434=1149.843,138.518,-56.936,-178.772,6.809,148.898
C04435=1149.848,138.269,-56.916,-178.775,6.807,148.898
C04436=1149.853,138.019,-56.895,-178.778,6.805,148.899
C04437=1149.857,137.770,-56.875,-178.780,6.804,148.899
C04438=1149.862,137.522,-56.855,-178.783,6.802,148.900
C04439=1149.867,137.273,-56.834,-178.786,6.800,148.900
C04440=1149.872,137.023,-56.814,-178.788,6.798,148.900
C04441=1149.877,136.774,-56.794,-178.791,6.796,148.900
C04442=1149.881,136.525,-56.773,-178.794,6.795,148.901
C04443=1149.886,136.276,-56.754,-178.796,6.793,148.901
C04444=1149.891,136.027,-56.733,-178.799,6.791,148.902
C04445=1149.896,135.778,-56.712,-178.802,6.789,148.902
C04446=1149.900,135.529,-56.692,-178.805,6.787,148.902
C04447=1149.905,135.279,-56.672,-178.808,6.785,148.903
C04448=1149.911,135.030,-56.652,-178.810,6.784,148.903
C04449=1149.915,134.782,-56.631,-178.813,6.782,148.904
C04450=1149.920,134.532,-56.612,-178.816,6.781,148.904
C04451=1149.924,134.283,-56.591,-178.819,6.779,148.905
C04452=1149.929,134.033,-56.571,-178.822,6.777,148.905
C04453=1149.934,133.784,-56.551,-178.824,6.775,148.905
C04454=1149.938,133.535,-56.530,-178.827,6.774,148.906
C04455=1149.944,133.286,-56.511,-178.830,6.772,148.906
C04456=1149.948,133.037,-56.490,-178.833,6.770,148.907
C04457=1149.953,132.788,-56.471,-178.835,6.769,148.907
C04458=1149.957,132.539,-56.450,-178.838,6.767,148.907
C04459=1149.962,132.289,-56.431,-178.841,6.765,148.908
C04460=1149.968,132.021,-56.408,-178.844,6.763,148.908
C04461=1149.972,131.752,-56.387,-178.847,6.761,148.909
C04462=1149.978,131.483,-56.366,-178.849,6.759,148.909
C04463=1149.983,131.215,-56.344,-178.853,6.757,148.909
C04464=1149.988,130.967,-56.325,-178.856,6.755,148.910
C04465=1149.992,130.718,-56.304,-178.858,6.753,148.910
C04466=1149.997,130.468,-56.285,-178.861,6.752,148.910
C04467=1150.002,130.219,-56.264,-178.864,6.750,148.911
C04468=1150.006,129.969,-56.244,-178.867,6.748,148.911
C04469=1150.012,129.720,-56.225,-178.870,6.747,148.912
C04470=1150.017,129.471,-56.204,-178.872,6.745,148.912
C04471=1150.022,129.222,-56.185,-178.875,6.743,148.913
C04472=1150.026,128.973,-56.164,-178.878,6.742,148.913
C04473=1150.031,128.724,-56.145,-178.880,6.740,148.913
C04474=1150.036,128.474,-56.125,-178.883,6.738,148.914
C04475=1150.041,128.225,-56.105,-178.886,6.737,148.914
C04476=1150.045,127.976,-56.085,-178.889,6.735,148.915
C04477=1150.051,127.727,-56.066,-178.891,6.733,148.915
C04478=1150.055,127.478,-56.046,-178.894,6.731,148.915
C04479=1150.060,127.228,-56.026,-178.897,6.730,148.916
C04480=1150.065,126.979,-56.006,-178.899,6.728,148.916
C04481=1150.069,126.731,-55.987,-178.902,6.726,148.917
C04482=1150.074,126.481,-55.967,-178.905,6.725,148.917
C04483=1150.078,126.232,-55.948,-178.908,6.723,148.917
C04484=1150.084,125.983,-55.928,-178.910,6.721,148.918
C04485=1150.088,125.734,-55.908,-178.913,6.719,148.918
C04486=1150.093,125.484,-55.888,-178.916,6.718,148.919
C04487=1150.098,125.235,-55.869,-178.919,6.716,148.919
C04488=1150.103,124.986,-55.849,-178.922,6.715,148.920
C04489=1150.107,124.737,-55.829,-178.924,6.713,148.920
C04490=1150.112,124.488,-55.809,-178.927,6.711,148.920
C04491=1150.118,124.239,-55.790,-178.930,6.710,148.921
C04492=1150.122,123.989,-55.771,-178.933,6.708,148.921
C04493=1150.126,123.740,-55.751,-178.935,6.706,148.922
C04494=1150.132,123.491,-55.732,-178.938,6.704,148.922
C04495=1150.136,123.242,-55.712,-178.941,6.703,148.922
C04496=1150.141,122.992,-55.692,-178.943,6.701,148.923
C04497=1150.146,122.744,-55.673,-178.946,6.699,148.923
C04498=1150.150,122.494,-55.654,-178.949,6.698,148.924
C04499=1150.156,122.245,-55.634,-178.952,6.696,148.924
C04500=1150.160,121.996,-55.615,-178.955,6.695,148.925
C04501=1150.165,121.746,-55.595,-178.957,6.693,148.925
C04502=1150.170,121.497,-55.576,-178.960,6.691,148.925
C04503=1150.174,121.248,-55.557,-178.963,6.689,148.926
C04504=1150.179,120.999,-55.537,-178.966,6.688,148.926
C04505=1150.184,120.750,-55.518,-178.968,6.686,148.927
C04506=1150.189,120.500,-55.498,-178.971,6.684,148.927
C04507=1150.195,120.251,-55.479,-178.974,6.683,148.927
C04508=1150.199,120.002,-55.460,-178.977,6.681,148.928
C04509=1150.204,119.753,-55.440,-178.979,6.679,148.928
C04510=1150.209,119.504,-55.421,-178.982,6.678,148.929
C04511=1150.213,119.254,-55.402,-178.985,6.676,148.929
C04512=1150.218,119.005,-55.382,-178.988,6.675,148.930
C04513=1150.223,118.756,-55.363,-178.990,6.674,148.930
C04514=1150.228,118.507,-55.343,-178.993,6.672,148.931
C04515=1150.232,118.258,-55.324,-178.995,6.670,148.931
C04516=1150.237,118.009,-55.305,-178.998,6.669,148.931
C04517=1150.242,117.759,-55.285,-179.001,6.667,148.932
C04518=1150.247,117.511,-55.267,-179.004,6.665,148.932
C04519=1150.252,117.261,-55.247,-179.007,6.664,148.933
C04520=1150.257,117.011,-55.228,-179.010,6.662,148.933
C04521=1150.261,116.762,-55.209,-179.012,6.660,148.934
C04522=1150.266,116.513,-55.190,-179.015,6.659,148.934
C04523=1150.271,116.264,-55.170,-179.018,6.657,148.934
C04524=1150.275,116.015,-55.151,-179.020,6.655,148.935
C04525=1150.281,115.766,-55.132,-179.023,6.654,148.935
C04526=1150.286,115.516,-55.113,-179.026,6.652,148.936
C04527=1150.290,115.267,-55.094,-179.029,6.651,148.936
C04528=1150.295,115.018,-55.075,-179.032,6.649,148.937
C04529=1150.300,114.769,-55.056,-179.034,6.648,148.937
C04530=1150.305,114.520,-55.038,-179.037,6.646,148.937
C04531=1150.310,114.270,-55.018,-179.039,6.645,148.938
C04532=1150.315,114.021,-54.999,-179.042,6.643,148.938
C04533=1150.319,113.772,-54.980,-179.045,6.641,148.939
C04534=1150.324,113.523,-54.962,-179.048,6.640,148.939
C04535=1150.329,113.273,-54.942,-179.051,6.638,148.940
C04536=1150.334,113.025,-54.923,-179.053,6.636,148.940
C04537=1150.339,112.774,-54.904,-179.056,6.635,148.941
C04538=1150.343,112.526,-54.886,-179.059,6.633,148.941
C04539=1150.348,112.276,-54.866,-179.062,6.631,148.941
C04540=1150.353,112.027,-54.848,-179.064,6.630,148.942
C04541=1150.358,111.778,-54.829,-179.067,6.629,148.942
C04542=1150.362,111.529,-54.810,-179.070,6.627,148.943
C04543=1150.368,111.279,-54.791,-179.072,6.626,148.943
C04544=1150.372,111.030,-54.772,-179.075,6.624,148.944
C04545=1150.378,110.781,-54.753,-179.078,6.622,148.944
C04546=1150.382,110.532,-54.735,-179.081,6.621,148.944
C04547=1150.387,110.283,-54.715,-179.083,6.619,148.945
C04548=1150.392,110.033,-54.697,-179.087,6.618,148.945
C04549=1150.397,109.784,-54.677,-179.089,6.616,148.946
C04550=1150.401,109.535,-54.659,-179.091,6.615,148.946
C04551=1150.407,109.286,-54.640,-179.094,6.613,148.947
C04552=1150.411,109.036,-54.622,-179.097,6.612,148.947
C04553=1150.416,108.787,-54.603,-179.100,6.610,148.947
C04554=1150.421,108.538,-54.584,-179.103,6.609,148.948
C04555=1150.425,108.289,-54.565,-179.106,6.607,148.949
C04556=1150.431,108.039,-54.547,-179.108,6.605,148.949
C04557=1150.435,107.790,-54.528,-179.111,6.604,148.949
C04558=1150.440,107.541,-54.510,-179.113,6.603,148.950
C04559=1150.445,107.292,-54.491,-179.116,6.601,148.950
C04560=1150.450,107.042,-54.472,-179.119,6.600,148.951
C04561=1150.455,106.792,-54.454,-179.122,6.598,148.951
C04562=1150.460,106.544,-54.435,-179.124,6.596,148.952
C04563=1150.464,106.294,-54.417,-179.127,6.595,148.952
C04564=1150.470,106.026,-54.396,-179.130,6.593,148.952
C04565=1150.475,105.758,-54.376,-179.133,6.592,148.953
C04566=1150.481,105.489,-54.356,-179.136,6.590,148.953
C04567=1150.486,105.221,-54.337,-179.139,6.589,148.954
C04568=1150.490,104.972,-54.318,-179.142,6.587,148.955
C04569=1150.495,104.722,-54.299,-179.145,6.585,148.955
C04570=1150.500,104.473,-54.281,-179.147,6.583,148.955
C04571=1150.504,104.224,-54.262,-179.149,6.583,148.956
C04572=1150.510,103.974,-54.244,-179.152,6.581,148.956
C04573=1150.515,103.725,-54.226,-179.155,6.580,148.957
C04574=1150.519,103.477,-54.207,-179.158,6.578,148.957
C04575=1150.524,103.227,-54.189,-179.161,6.576,148.958
C04576=1150.529,102.977,-54.170,-179.164,6.574,148.958
C04577=1150.534,102.728,-54.152,-179.166,6.574,148.958
C04578=1150.539,102.480,-54.134,-179.169,6.572,148.959
C04579=1150.543,102.230,-54.115,-179.172,6.571,148.960
C04580=1150.549,101.980,-54.097,-179.174,6.569,148.960
C04581=1150.554,101.731,-54.079,-179.177,6.567,148.960
C04582=1150.559,101.482,-54.061,-179.180,6.566,148.961
C04583=1150.563,101.233,-54.042,-179.182,6.565,148.961
C04584=1150.568,100.983,-54.024,-179.185,6.563,148.962
C04585=1150.573,100.734,-54.005,-179.188,6.562,148.962
C04586=1150.578,100.485,-53.987,-179.191,6.560,148.963
C04587=1150.583,100.236,-53.969,-179.194,6.559,148.963
C04588=1150.587,99.986,-53.951,-179.196,6.558,148.964
C04589=1150.592,99.737,-53.933,-179.199,6.556,148.964
C04590=1150.597,99.488,-53.914,-179.201,6.554,148.965
C04591=1150.602,99.239,-53.896,-179.204,6.553,148.965
C04592=1150.607,98.989,-53.877,-179.207,6.551,148.966
C04593=1150.612,98.739,-53.859,-179.209,6.550,148.966
C04594=1150.617,98.490,-53.841,-179.212,6.549,148.966
C04595=1150.622,98.241,-53.823,-179.215,6.547,148.967
C04596=1150.627,97.992,-53.805,-179.218,6.545,148.967
C04597=1150.631,97.743,-53.787,-179.221,6.544,148.968
C04598=1150.636,97.494,-53.769,-179.223,6.543,148.968
C04599=1150.641,97.244,-53.751,-179.226,6.541,148.969
C04600=1150.646,96.994,-53.733,-179.228,6.540,148.969
C04601=1150.650,96.745,-53.715,-179.232,6.538,148.970
C04602=1150.655,96.496,-53.697,-179.234,6.537,148.970
C04603=1150.661,96.247,-53.678,-179.237,6.536,148.971
C04604=1150.666,95.997,-53.660,-179.239,6.534,148.971
C04605=1150.671,95.748,-53.642,-179.243,6.533,148.972
C04606=1150.675,95.498,-53.624,-179.245,6.531,148.972
C04607=1150.680,95.249,-53.606,-179.248,6.530,148.973
C04608=1150.685,95.000,-53.588,-179.250,6.529,148.973
C04609=1150.690,94.751,-53.570,-179.253,6.527,148.973
C04610=1150.695,94.501,-53.553,-179.256,6.526,148.974
C04611=1150.700,94.252,-53.535,-179.259,6.524,148.974
C04612=1150.705,94.003,-53.517,-179.261,6.523,148.975
C04613=1150.710,93.754,-53.499,-179.264,6.521,148.975
C04614=1150.715,93.504,-53.481,-179.267,6.520,148.976
C04615=1150.720,93.255,-53.463,-179.270,6.518,148.976
C04616=1150.725,93.006,-53.445,-179.272,6.518,148.977
C04617=1150.730,92.756,-53.428,-179.274,6.516,148.977
C04618=1150.733,92.507,-53.410,-179.278,6.515,148.978
C04619=1150.738,92.258,-53.392,-179.280,6.513,148.978
C04620=1150.743,92.008,-53.374,-179.283,6.511,148.979
C04621=1150.748,91.759,-53.356,-179.285,6.510,148.979
C04622=1150.753,91.509,-53.339,-179.289,6.509,148.980
C04623=1150.758,91.260,-53.321,-179.291,6.507,148.980
C04624=1150.763,91.011,-53.303,-179.294,6.506,148.981
C04625=1150.768,90.762,-53.285,-179.296,6.505,148.981
C04626=1150.773,90.512,-53.268,-179.299,6.503,148.982
C04627=1150.778,90.263,-53.250,-179.302,6.502,148.982
C04628=1150.783,90.014,-53.232,-179.304,6.501,148.982
C04629=1150.787,89.765,-53.214,-179.307,6.499,148.983
C04630=1150.793,89.515,-53.197,-179.310,6.498,148.984
C04631=1150.797,89.266,-53.179,-179.313,6.496,148.984
C04632=1150.802,89.017,-53.161,-179.315,6.495,148.984
C04633=1150.808,88.767,-53.144,-179.318,6.494,148.985
C04634=1150.812,88.518,-53.126,-179.321,6.492,148.985
C04635=1150.817,88.269,-53.108,-179.324,6.491,148.986
C04636=1150.822,88.019,-53.091,-179.326,6.490,148.986
C04637=1150.827,87.770,-53.073,-179.329,6.488,148.987
C04638=1150.832,87.520,-53.056,-179.332,6.487,148.987
C04639=1150.837,87.271,-53.038,-179.334,6.486,148.988
C04640=1150.841,87.022,-53.020,-179.337,6.484,148.988
C04641=1150.846,86.772,-53.003,-179.340,6.483,148.989
C04642=1150.851,86.523,-52.985,-179.343,6.481,148.989
C04643=1150.856,86.273,-52.968,-179.345,6.480,148.990
C04644=1150.861,86.024,-52.950,-179.348,6.479,148.990
C04645=1150.866,85.775,-52.934,-179.351,6.477,148.991
C04646=1150.871,85.526,-52.916,-179.353,6.476,148.991
C04647=1150.877,85.276,-52.898,-179.356,6.475,148.992
C04648=1150.881,85.027,-52.881,-179.359,6.473,148.992
C04649=1150.886,84.778,-52.863,-179.362,6.472,148.993
C04650=1150.891,84.529,-52.846,-179.364,6.471,148.993
C04651=1150.896,84.279,-52.829,-179.366,6.469,148.994
C04652=1150.900,84.030,-52.811,-179.370,6.468,148.994
C04653=1150.905,83.780,-52.794,-179.372,6.467,148.995
C04654=1150.910,83.531,-52.776,-179.375,6.465,148.995
C04655=1150.915,83.281,-52.759,-179.378,6.464,148.996
C04656=1150.920,83.033,-52.742,-179.380,6.463,148.996
C04657=1150.926,82.783,-52.724,-179.383,6.462,148.997
C04658=1150.930,82.534,-52.707,-179.386,6.460,148.997
C04659=1150.935,82.284,-52.690,-179.389,6.459,148.998
C04660=1150.940,82.035,-52.672,-179.391,6.458,148.998
C04661=1150.944,81.786,-52.655,-179.394,6.456,148.998
C04662=1150.950,81.536,-52.638,-179.397,6.455,148.999
C04663=1150.955,81.286,-52.621,-179.399,6.454,149.000
C04664=1150.960,81.038,-52.604,-179.402,6.452,149.000
C04665=1150.965,80.788,-52.586,-179.405,6.451,149.001
C04666=1150.969,80.539,-52.570,-179.407,6.450,149.001
C04667=1150.974,80.290,-52.552,-179.410,6.448,149.001
C04668=1150.980,80.021,-52.533,-179.413,6.447,149.002
C04669=1150.985,79.753,-52.515,-179.416,6.445,149.003
C04670=1150.990,79.484,-52.497,-179.419,6.444,149.003
C04671=1150.996,79.216,-52.478,-179.421,6.443,149.004
C04672=1151.000,78.967,-52.461,-179.424,6.441,149.004
C04673=1151.006,78.717,-52.444,-179.427,6.440,149.005
C04674=1151.010,78.468,-52.427,-179.429,6.439,149.005
C04675=1151.015,78.218,-52.410,-179.432,6.438,149.006
C04676=1151.020,77.970,-52.393,-179.435,6.436,149.006
C04677=1151.025,77.720,-52.375,-179.437,6.435,149.007
C04678=1151.030,77.470,-52.359,-179.440,6.434,149.007
C04679=1151.035,77.221,-52.341,-179.443,6.432,149.008
C04680=1151.039,76.971,-52.325,-179.445,6.432,149.008
C04681=1151.045,76.722,-52.308,-179.448,6.430,149.009
C04682=1151.049,76.473,-52.290,-179.451,6.429,149.009
C04683=1151.055,76.223,-52.273,-179.453,6.428,149.010
C04684=1151.059,75.974,-52.256,-179.456,6.426,149.010
C04685=1151.065,75.725,-52.240,-179.459,6.425,149.011
C04686=1151.069,75.475,-52.223,-179.462,6.424,149.011
C04687=1151.075,75.226,-52.206,-179.464,6.422,149.012
C04688=1151.079,74.976,-52.189,-179.467,6.422,149.012
C04689=1151.085,74.727,-52.172,-179.470,6.420,149.013
C04690=1151.089,74.478,-52.155,-179.472,6.418,149.013
C04691=1151.094,74.229,-52.138,-179.475,6.418,149.014
C04692=1151.099,73.980,-52.121,-179.478,6.416,149.014
C04693=1151.104,73.730,-52.104,-179.481,6.415,149.015
C04694=1151.109,73.480,-52.087,-179.483,6.414,149.015
C04695=1151.114,73.231,-52.071,-179.486,6.412,149.016
C04696=1151.119,72.982,-52.054,-179.488,6.412,149.016
C04697=1151.124,72.732,-52.037,-179.491,6.410,149.017
C04698=1151.128,72.483,-52.020,-179.494,6.409,149.017
C04699=1151.134,72.234,-52.003,-179.496,6.408,149.018
C04700=1151.139,71.984,-51.987,-179.499,6.406,149.018
C04701=1151.143,71.735,-51.970,-179.502,6.406,149.019
C04702=1151.149,71.486,-51.953,-179.504,6.404,149.019
C04703=1151.153,71.236,-51.936,-179.508,6.403,149.020
C04704=1151.158,70.987,-51.920,-179.510,6.402,149.020
C04705=1151.164,70.737,-51.903,-179.512,6.400,149.021
C04706=1151.169,70.487,-51.887,-179.515,6.400,149.021
C04707=1151.173,70.238,-51.870,-179.518,6.398,149.022
C04708=1151.179,69.989,-51.853,-179.521,6.396,149.022
C04709=1151.183,69.739,-51.837,-179.523,6.396,149.023
C04710=1151.188,69.490,-51.820,-179.526,6.394,149.023
C04711=1151.194,69.241,-51.803,-179.528,6.393,149.024
C04712=1151.198,68.991,-51.786,-179.531,6.392,149.024
C04713=1151.203,68.742,-51.770,-179.534,6.390,149.025
C04714=1151.208,68.492,-51.754,-179.536,6.389,149.025
C04715=1151.213,68.243,-51.737,-179.539,6.388,149.026
C04716=1151.218,67.994,-51.721,-179.542,6.387,149.026
C04717=1151.223,67.744,-51.704,-179.544,6.386,149.027
C04718=1151.227,67.495,-51.687,-179.548,6.384,149.027
C04719=1151.233,67.245,-51.671,-179.550,6.383,149.028
C04720=1151.238,66.996,-51.654,-179.552,6.382,149.028
C04721=1151.243,66.747,-51.638,-179.555,6.381,149.029
C04722=1151.247,66.497,-51.622,-179.558,6.380,149.029
C04723=1151.252,66.248,-51.605,-179.560,6.379,149.030
C04724=1151.258,65.998,-51.589,-179.563,6.377,149.031
C04725=1151.263,65.749,-51.572,-179.566,6.376,149.031
C04726=1151.268,65.500,-51.556,-179.569,6.375,149.032
C04727=1151.272,65.250,-51.540,-179.571,6.374,149.032
C04728=1151.277,65.001,-51.523,-179.573,6.373,149.033
C04729=1151.283,64.751,-51.506,-179.577,6.371,149.033
C04730=1151.287,64.502,-51.489,-179.579,6.371,149.034
C04731=1151.293,64.252,-51.474,-179.582,6.369,149.034
C04732=1151.297,64.003,-51.457,-179.584,6.368,149.035
C04733=1151.302,63.754,-51.441,-179.587,6.367,149.035
C04734=1151.307,63.504,-51.425,-179.590,6.365,149.036
C04735=1151.312,63.255,-51.409,-179.592,6.365,149.036
C04736=1151.317,63.005,-51.392,-179.595,6.363,149.037
C04737=1151.323,62.756,-51.376,-179.598,6.362,149.037
C04738=1151.327,62.506,-51.359,-179.600,6.361,149.038
C04739=1151.332,62.257,-51.344,-179.603,6.360,149.038
C04740=1151.337,62.008,-51.327,-179.606,6.359,149.039
C04741=1151.342,61.758,-51.311,-179.608,6.358,149.039
C04742=1151.347,61.509,-51.295,-179.611,6.356,149.040
C04743=1151.352,61.260,-51.278,-179.613,6.356,149.040
C04744=1151.357,61.010,-51.262,-179.616,6.354,149.041
C04745=1151.362,60.761,-51.246,-179.619,6.353,149.042
C04746=1151.367,60.511,-51.230,-179.621,6.352,149.042
C04747=1151.372,60.262,-51.214,-179.624,6.350,149.042
C04748=1151.376,60.012,-51.198,-179.627,6.350,149.043
C04749=1151.381,59.763,-51.182,-179.630,6.348,149.043
C04750=1151.386,59.513,-51.166,-179.632,6.347,149.044
C04751=1151.391,59.264,-51.149,-179.635,6.346,149.045
C04752=1151.397,59.015,-51.134,-179.637,6.345,149.045
C04753=1151.401,58.766,-51.117,-179.640,6.344,149.046
C04754=1151.407,58.516,-51.101,-179.643,6.343,149.046
C04755=1151.411,58.266,-51.086,-179.645,6.341,149.047
C04756=1151.416,58.017,-51.069,-179.648,6.341,149.047
C04757=1151.421,57.767,-51.053,-179.651,6.339,149.048
C04758=1151.426,57.518,-51.037,-179.653,6.339,149.048
C04759=1151.432,57.269,-51.021,-179.656,6.337,149.049
C04760=1151.436,57.019,-51.005,-179.658,6.336,149.049
C04761=1151.442,56.770,-50.989,-179.661,6.335,149.050
C04762=1151.446,56.520,-50.973,-179.664,6.334,149.050
C04763=1151.451,56.271,-50.957,-179.666,6.332,149.051
C04764=1151.457,56.022,-50.941,-179.669,6.332,149.051
C04765=1151.462,55.772,-50.925,-179.672,6.330,149.052
C04766=1151.467,55.523,-50.909,-179.674,6.330,149.053
C04767=1151.471,55.273,-50.893,-179.677,6.328,149.053
C04768=1151.477,55.023,-50.877,-179.679,6.327,149.053
C04769=1151.482,54.775,-50.861,-179.682,6.326,149.054
C04770=1151.487,54.524,-50.845,-179.685,6.325,149.055
C04771=1151.492,54.275,-50.830,-179.688,6.324,149.055
C04772=1151.497,54.007,-50.813,-179.690,6.323,149.056
C04773=1151.502,53.738,-50.796,-179.693,6.322,149.056
C04774=1151.507,53.469,-50.779,-179.696,6.320,149.057
C04775=1151.513,53.201,-50.762,-179.699,6.319,149.057
C04776=1151.518,52.951,-50.746,-179.701,6.318,149.058
C04777=1151.523,52.702,-50.730,-179.704,6.317,149.059
C04778=1151.528,52.452,-50.714,-179.707,6.316,149.059
C04779=1151.534,52.203,-50.698,-179.709,6.315,149.060
C04780=1151.538,51.953,-50.683,-179.712,6.314,149.060
C04781=1151.543,51.704,-50.667,-179.714,6.313,149.060
C04782=1151.548,51.454,-50.652,-179.718,6.311,149.061
C04783=1151.554,51.206,-50.636,-179.720,6.311,149.062
C04784=1151.558,50.956,-50.620,-179.723,6.309,149.062
C04785=1151.563,50.707,-50.605,-179.725,6.308,149.063
C04786=1151.568,50.457,-50.589,-179.728,6.307,149.063
C04787=1151.573,50.207,-50.573,-179.731,6.306,149.064
C04788=1151.579,49.958,-50.557,-179.733,6.305,149.064
C04789=1151.583,49.709,-50.542,-179.736,6.304,149.065
C04790=1151.588,49.459,-50.526,-179.739,6.303,149.065
C04791=1151.593,49.210,-50.510,-179.741,6.302,149.066
C04792=1151.598,48.960,-50.495,-179.743,6.301,149.066
C04793=1151.603,48.711,-50.480,-179.746,6.300,149.067
C04794=1151.608,48.461,-50.464,-179.749,6.299,149.068
C04795=1151.613,48.212,-50.448,-179.752,6.297,149.068
C04796=1151.619,47.962,-50.432,-179.754,6.297,149.068
C04797=1151.623,47.713,-50.417,-179.757,6.295,149.069
C04798=1151.628,47.463,-50.402,-179.759,6.294,149.070
C04799=1151.633,47.214,-50.386,-179.762,6.293,149.070
C04800=1151.638,46.965,-50.371,-179.765,6.292,149.071
C04801=1151.644,46.715,-50.355,-179.767,6.292,149.071
C04802=1151.648,46.465,-50.339,-179.770,6.290,149.072
C04803=1151.653,46.216,-50.324,-179.772,6.289,149.072
C04804=1151.658,45.967,-50.309,-179.775,6.288,149.073
C04805=1151.664,45.717,-50.293,-179.777,6.287,149.073
C04806=1151.668,45.467,-50.278,-179.781,6.286,149.074
C04807=1151.673,45.218,-50.262,-179.783,6.285,149.075
C04808=1151.679,44.969,-50.247,-179.785,6.284,149.075
C04809=1151.683,44.719,-50.232,-179.788,6.283,149.076
C04810=1151.689,44.470,-50.216,-179.790,6.282,149.076
C04811=1151.693,44.220,-50.201,-179.794,6.281,149.077
C04812=1151.698,43.970,-50.186,-179.796,6.280,149.077
C04813=1151.704,43.721,-50.170,-179.799,6.279,149.078
C04814=1151.708,43.472,-50.155,-179.801,6.278,149.078
C04815=1151.714,43.222,-50.140,-179.803,6.277,149.079
C04816=1151.718,42.973,-50.125,-179.807,6.276,149.079
C04817=1151.723,42.723,-50.109,-179.809,6.275,149.080
C04818=1151.729,42.474,-50.093,-179.812,6.274,149.081
C04819=1151.734,42.224,-50.079,-179.814,6.273,149.081
C04820=1151.739,41.975,-50.063,-179.817,6.272,149.082
C04821=1151.744,41.726,-50.048,-179.820,6.271,149.082
C04822=1151.749,41.476,-50.033,-179.822,6.270,149.083
C04823=1151.754,41.227,-50.018,-179.825,6.269,149.083
C04824=1151.759,40.976,-50.003,-179.827,6.268,149.084
C04825=1151.763,40.727,-49.988,-179.830,6.267,149.084
C04826=1151.769,40.478,-49.972,-179.833,6.266,149.085
C04827=1151.773,40.229,-49.957,-179.835,6.265,149.085
C04828=1151.779,39.979,-49.942,-179.838,6.263,149.086
C04829=1151.784,39.730,-49.927,-179.840,6.263,149.086
C04830=1151.789,39.480,-49.911,-179.843,6.262,149.087
C04831=1151.794,39.231,-49.896,-179.845,6.261,149.087
C04832=1151.799,38.981,-49.882,-179.848,6.260,149.088
C04833=1151.803,38.731,-49.866,-179.850,6.259,149.089
C04834=1151.809,38.482,-49.851,-179.854,6.258,149.089
C04835=1151.814,38.232,-49.836,-179.856,6.257,149.090
C04836=1151.819,37.983,-49.821,-179.858,6.255,149.090
C04837=1151.824,37.734,-49.806,-179.861,6.255,149.091
C04838=1151.830,37.484,-49.791,-179.863,6.254,149.091
C04839=1151.834,37.235,-49.776,-179.866,6.253,149.092
C04840=1151.840,36.985,-49.760,-179.869,6.252,149.092
C04841=1151.845,36.735,-49.746,-179.871,6.252,149.093
C04842=1151.849,36.486,-49.731,-179.874,6.250,149.094
C04843=1151.855,36.236,-49.716,-179.877,6.249,149.094
C04844=1151.860,35.987,-49.701,-179.879,6.248,149.095
C04845=1151.865,35.738,-49.686,-179.882,6.247,149.095
C04846=1151.870,35.488,-49.671,-179.884,6.247,149.096
C04847=1151.875,35.239,-49.656,-179.887,6.245,149.096
C04848=1151.880,34.989,-49.641,-179.890,6.244,149.097
C04849=1151.885,34.740,-49.627,-179.892,6.244,149.097
C04850=1151.891,34.490,-49.612,-179.895,6.242,149.098
C04851=1151.895,34.241,-49.597,-179.897,6.241,149.098
C04852=1151.900,33.991,-49.582,-179.900,6.241,149.099
C04853=1151.906,33.742,-49.567,-179.903,6.239,149.100
C04854=1151.911,33.492,-49.552,-179.905,6.239,149.100
C04855=1151.915,33.243,-49.538,-179.907,6.238,149.101
C04856=1151.921,32.993,-49.523,-179.910,6.236,149.101
C04857=1151.926,32.744,-49.508,-179.913,6.236,149.102
C04858=1151.930,32.494,-49.493,-179.916,6.234,149.102
C04859=1151.936,32.245,-49.478,-179.918,6.234,149.103
C04860=1151.941,31.995,-49.463,-179.920,6.233,149.103
C04861=1151.945,31.746,-49.449,-179.924,6.232,149.104
C04862=1151.950,31.496,-49.434,-179.926,6.231,149.105
C04863=1151.956,31.246,-49.419,-179.928,6.230,149.105
C04864=1151.961,30.997,-49.404,-179.931,6.229,149.106
C04865=1151.966,30.747,-49.390,-179.933,6.228,149.106
C04866=1151.971,30.498,-49.374,-179.936,6.227,149.107
C04867=1151.976,30.248,-49.360,-179.939,6.226,149.107
C04868=1151.981,29.999,-49.346,-179.941,6.225,149.108
C04869=1151.986,29.749,-49.331,-179.944,6.225,149.108
C04870=1151.991,29.499,-49.316,-179.946,6.224,149.109
C04871=1151.996,29.250,-49.302,-179.949,6.222,149.110
C04872=1152.001,29.001,-49.287,-179.952,6.222,149.110
C04873=1152.006,28.751,-49.273,-179.954,6.221,149.111
C04874=1152.011,28.501,-49.258,-179.957,6.220,149.111
C04875=1152.016,28.252,-49.243,-179.959,6.219,149.112
C04876=1152.022,27.984,-49.227,-179.962,6.218,149.112
C04877=1152.027,27.714,-49.212,-179.965,6.217,149.113
C04878=1152.033,27.446,-49.197,-179.968,6.216,149.114
C04879=1152.038,27.176,-49.180,-179.971,6.215,149.114
C04880=1152.043,26.927,-49.166,-179.973,6.214,149.115
C04881=1152.048,26.677,-49.152,-179.975,6.213,149.115
C04882=1152.053,26.428,-49.137,-179.978,6.212,149.116
C04883=1152.058,26.178,-49.123,-179.980,6.211,149.116
C04884=1152.064,25.928,-49.108,-179.984,6.210,149.117
C04885=1152.069,25.679,-49.094,-179.986,6.209,149.117
C04886=1152.074,25.430,-49.079,-179.988,6.209,149.118
C04887=1152.079,25.180,-49.064,-179.990,6.208,149.119
C04888=1152.084,24.931,-49.050,-179.994,6.207,149.119
C04889=1152.089,24.681,-49.036,-179.996,6.206,149.120
C04890=1152.094,24.431,-49.022,-179.999,6.206,149.120
C04891=1152.099,24.181,-49.007,179.999,6.204,149.121
C04892=1152.104,23.933,-48.993,179.997,6.203,149.121
C04893=1152.110,23.683,-48.978,179.994,6.203,149.122
C04894=1152.114,23.433,-48.964,179.992,6.202,149.122
C04895=1152.119,23.184,-48.949,179.988,6.201,149.123
C04896=1152.124,22.934,-48.935,179.986,6.200,149.124
C04897=1152.129,22.684,-48.921,179.984,6.199,149.124
C04898=1152.135,22.435,-48.907,179.981,6.198,149.125
C04899=1152.140,22.186,-48.893,179.978,6.197,149.125
C04900=1152.144,21.936,-48.878,179.976,6.196,149.126
C04901=1152.149,21.687,-48.863,179.973,6.196,149.127
C04902=1152.154,21.437,-48.849,179.971,6.194,149.127
C04903=1152.160,21.188,-48.835,179.968,6.194,149.128
C04904=1152.165,20.938,-48.821,179.966,6.193,149.128
C04905=1152.170,20.689,-48.807,179.963,6.192,149.129
C04906=1152.175,20.439,-48.792,179.960,6.191,149.129
C04907=1152.180,20.189,-48.778,179.958,6.190,149.130
C04908=1152.185,19.940,-48.764,179.956,6.190,149.130
C04909=1152.190,19.690,-48.750,179.953,6.189,149.131
C04910=1152.195,19.441,-48.736,179.950,6.187,149.132
C04911=1152.200,19.191,-48.721,179.948,6.187,149.132
C04912=1152.206,18.942,-48.707,179.945,6.186,149.133
C04913=1152.211,18.692,-48.693,179.943,6.185,149.133
C04914=1152.216,18.443,-48.679,179.940,6.184,149.134
C04915=1152.221,18.193,-48.664,179.938,6.183,149.134
C04916=1152.226,17.944,-48.651,179.935,6.183,149.135
C04917=1152.231,17.694,-48.636,179.932,6.181,149.135
C04918=1152.236,17.444,-48.622,179.930,6.181,149.136
C04919=1152.241,17.194,-48.608,179.928,6.180,149.137
C04920=1152.247,16.945,-48.595,179.925,6.179,149.137
C04921=1152.251,16.696,-48.581,179.923,6.179,149.138
C04922=1152.256,16.446,-48.567,179.920,6.177,149.138
C04923=1152.262,16.197,-48.553,179.917,6.177,149.139
C04924=1152.267,15.947,-48.538,179.915,6.176,149.139
C04925=1152.272,15.698,-48.524,179.913,6.175,149.140
C04926=1152.276,15.448,-48.510,179.910,6.174,149.140
C04927=1152.282,15.198,-48.497,179.907,6.173,149.141
C04928=1152.287,14.949,-48.482,179.905,6.172,149.142
C04929=1152.292,14.699,-48.468,179.902,6.172,149.142
C04930=1152.297,14.450,-48.455,179.900,6.170,149.143
C04931=1152.302,14.200,-48.441,179.897,6.170,149.143
C04932=1152.307,13.950,-48.427,179.895,6.169,149.144
C04933=1152.313,13.701,-48.413,179.892,6.169,149.145
C04934=1152.318,13.451,-48.399,179.890,6.168,149.145
C04935=1152.323,13.202,-48.384,179.887,6.167,149.146
C04936=1152.328,12.953,-48.371,179.884,6.166,149.146
C04937=1152.333,12.703,-48.358,179.882,6.165,149.147
C04938=1152.338,12.453,-48.343,179.880,6.164,149.147
C04939=1152.343,12.204,-48.329,179.876,6.163,149.148
C04940=1152.348,11.954,-48.315,179.874,6.162,149.148
C04941=1152.353,11.704,-48.302,179.872,6.162,149.149
C04942=1152.358,11.455,-48.288,179.869,6.161,149.150
C04943=1152.363,11.205,-48.274,179.867,6.161,149.150
C04944=1152.369,10.955,-48.260,179.864,6.159,149.151
C04945=1152.374,10.706,-48.247,179.862,6.158,149.151
C04946=1152.378,10.457,-48.233,179.859,6.158,149.152
C04947=1152.384,10.207,-48.220,179.857,6.157,149.152
C04948=1152.389,9.957,-48.205,179.854,6.156,149.153
C04949=1152.394,9.708,-48.191,179.852,6.155,149.153
C04950=1152.399,9.458,-48.178,179.849,6.154,149.154
C04951=1152.404,9.209,-48.164,179.847,6.154,149.155
C04952=1152.410,8.960,-48.150,179.844,6.153,149.155
C04953=1152.414,8.710,-48.137,179.842,6.152,149.156
C04954=1152.419,8.460,-48.123,179.839,6.152,149.156
C04955=1152.425,8.210,-48.110,179.836,6.150,149.157
C04956=1152.430,7.961,-48.096,179.834,6.150,149.158
C04957=1152.435,7.712,-48.082,179.832,6.149,149.158
C04958=1152.440,7.462,-48.069,179.829,6.148,149.159
C04959=1152.446,7.213,-48.055,179.827,6.148,149.159
C04960=1152.450,6.962,-48.042,179.824,6.146,149.160
C04961=1152.455,6.713,-48.028,179.821,6.146,149.160
C04962=1152.461,6.463,-48.014,179.819,6.145,149.161
C04963=1152.465,6.214,-48.001,179.817,6.144,149.162
C04964=1152.471,5.964,-47.987,179.814,6.144,149.162
C04965=1152.476,5.714,-47.973,179.812,6.143,149.163
C04966=1152.481,5.465,-47.961,179.809,6.142,149.163
C04967=1152.486,5.215,-47.946,179.806,6.141,149.164
C04968=1152.491,4.966,-47.934,179.804,6.141,149.165
C04969=1152.496,4.716,-47.919,179.802,6.140,149.165
C04970=1152.502,4.467,-47.906,179.799,6.139,149.165
C04971=1152.506,4.217,-47.893,179.797,6.138,149.166
C04972=1152.512,3.968,-47.879,179.794,6.137,149.167
C04973=1152.516,3.718,-47.866,179.791,6.136,149.167
C04974=1152.522,3.469,-47.852,179.789,6.136,149.168
C04975=1152.527,3.219,-47.838,179.786,6.135,149.168
C04976=1152.532,2.970,-47.826,179.784,6.134,149.169
C04977=1152.538,2.719,-47.812,179.782,6.134,149.170
C04978=1152.542,2.471,-47.799,179.779,6.132,149.170
C04979=1152.548,2.220,-47.785,179.776,6.132,149.171
C04980=1152.553,1.951,-47.770,179.774,6.131,149.171
C04981=1152.559,1.682,-47.757,179.771,6.131,149.172
C04982=1152.564,1.412,-47.742,179.768,6.129,149.173
C04983=1152.570,1.142,-47.728,179.765,6.129,149.173
C04984=1152.575,0.894,-47.714,179.763,6.128,149.174
C04985=1152.580,0.643,-47.701,179.761,6.128,149.174
C04986=1152.585,0.394,-47.688,179.758,6.127,149.175
C04987=1152.590,0.144,-47.674,179.756,6.126,149.176
C04988=1152.595,-0.105,-47.661,179.753,6.125,149.176
C04989=1152.601,-0.355,-47.648,179.751,6.124,149.176
C04990=1152.605,-0.604,-47.634,179.748,6.124,149.177
C04991=1152.611,-0.854,-47.621,179.746,6.123,149.178
C04992=1152.616,-1.104,-47.608,179.743,6.122,149.178
C04993=1152.621,-1.353,-47.594,179.741,6.121,149.179
C04994=1152.626,-1.603,-47.581,179.739,6.121,149.179
C04995=1152.632,-1.852,-47.568,179.736,6.119,149.180
C04996=1152.637,-2.102,-47.556,179.733,6.119,149.181
C04997=1152.642,-2.351,-47.541,179.731,6.118,149.181
C04998=1152.647,-2.601,-47.529,179.728,6.118,149.182
C04999=1152.652,-2.851,-47.515,179.726,6.117,149.182
C05000=1152.657,-3.100,-47.502,179.723,6.116,149.183
C05001=1152.662,-3.350,-47.490,179.721,6.116,149.183
C05002=1152.667,-3.599,-47.476,179.719,6.115,149.184
C05003=1152.672,-3.849,-47.463,179.716,6.114,149.185
C05004=1152.678,-4.099,-47.449,179.713,6.113,149.185
C05005=1152.683,-4.348,-47.437,179.711,6.112,149.186
C05006=1152.688,-4.598,-47.424,179.708,6.112,149.186
C05007=1152.693,-4.848,-47.411,179.706,6.111,149.187
C05008=1152.698,-5.097,-47.397,179.704,6.111,149.188
C05009=1152.704,-5.346,-47.384,179.701,6.110,149.188
C05010=1152.708,-5.596,-47.371,179.699,6.109,149.189
C05011=1152.713,-5.846,-47.359,179.697,6.109,149.189
C05012=1152.719,-6.096,-47.345,179.694,6.108,149.190
C05013=1152.724,-6.345,-47.332,179.691,6.107,149.190
C05014=1152.729,-6.595,-47.320,179.688,6.106,149.191
C05015=1152.734,-6.845,-47.306,179.686,6.105,149.191
C05016=1152.739,-7.094,-47.294,179.684,6.105,149.192
C05017=1152.744,-7.344,-47.281,179.681,6.104,149.193
C05018=1152.749,-7.593,-47.267,179.679,6.104,149.193
C05019=1152.755,-7.843,-47.254,179.677,6.103,149.194
C05020=1152.760,-8.092,-47.242,179.674,6.102,149.194
C05021=1152.765,-8.342,-47.228,179.672,6.102,149.195
C05022=1152.770,-8.592,-47.215,179.669,6.101,149.196
C05023=1152.775,-8.841,-47.203,179.667,6.100,149.196
C05024=1152.780,-9.090,-47.190,179.665,6.099,149.197
C05025=1152.786,-9.340,-47.177,179.661,6.098,149.197
C05026=1152.791,-9.590,-47.164,179.659,6.097,149.198
C05027=1152.796,-9.839,-47.151,179.657,6.097,149.198
C05028=1152.801,-10.089,-47.138,179.654,6.096,149.199
C05029=1152.806,-10.339,-47.125,179.652,6.096,149.200
C05030=1152.811,-10.588,-47.113,179.650,6.095,149.200
C05031=1152.816,-10.837,-47.100,179.647,6.095,149.201
C05032=1152.822,-11.088,-47.087,179.645,6.094,149.201
C05033=1152.827,-11.338,-47.075,179.642,6.093,149.202
C05034=1152.832,-11.587,-47.062,179.640,6.092,149.202
C05035=1152.837,-11.837,-47.049,179.637,6.092,149.203
C05036=1152.842,-12.086,-47.036,179.635,6.091,149.204
C05037=1152.848,-12.336,-47.023,179.632,6.091,149.204
C05038=1152.853,-12.585,-47.011,179.630,6.090,149.205
C05039=1152.857,-12.835,-46.998,179.628,6.090,149.205
C05040=1152.863,-13.085,-46.985,179.625,6.088,149.206
C05041=1152.868,-13.334,-46.973,179.622,6.088,149.207
C05042=1152.874,-13.584,-46.960,179.620,6.087,149.207
C05043=1152.878,-13.834,-46.947,179.617,6.086,149.208
C05044=1152.883,-14.084,-46.934,179.615,6.085,149.208
C05045=1152.889,-14.333,-46.922,179.613,6.085,149.209
C05046=1152.894,-14.582,-46.909,179.610,6.084,149.209
C05047=1152.899,-14.831,-46.897,179.608,6.084,149.210
C05048=1152.904,-15.082,-46.884,179.606,6.083,149.211
C05049=1152.910,-15.332,-46.871,179.603,6.083,149.211
C05050=1152.915,-15.581,-46.859,179.601,6.082,149.212
C05051=1152.920,-15.830,-46.846,179.598,6.081,149.212
C05052=1152.925,-16.080,-46.833,179.596,6.081,149.213
C05053=1152.930,-16.330,-46.821,179.593,6.080,149.214
C05054=1152.935,-16.580,-46.809,179.591,6.079,149.214
C05055=1152.940,-16.829,-46.796,179.588,6.079,149.215
C05056=1152.946,-17.079,-46.783,179.586,6.078,149.215
C05057=1152.951,-17.329,-46.771,179.584,6.077,149.216
C05058=1152.956,-17.578,-46.758,179.581,6.077,149.216
C05059=1152.961,-17.828,-46.745,179.579,6.076,149.217
C05060=1152.966,-18.077,-46.733,179.576,6.076,149.217
C05061=1152.971,-18.327,-46.721,179.574,6.075,149.218
C05062=1152.977,-18.576,-46.708,179.572,6.074,149.219
C05063=1152.982,-18.826,-46.696,179.569,6.074,149.219
C05064=1152.987,-19.076,-46.684,179.567,6.073,149.220
C05065=1152.992,-19.326,-46.671,179.565,6.072,149.220
C05066=1152.997,-19.575,-46.658,179.561,6.071,149.221
C05067=1153.002,-19.825,-46.646,179.559,6.070,149.221
C05068=1153.007,-20.074,-46.634,179.557,6.070,149.222
C05069=1153.012,-20.324,-46.621,179.554,6.069,149.223
C05070=1153.018,-20.574,-46.609,179.552,6.069,149.223
C05071=1153.023,-20.823,-46.597,179.549,6.068,149.224
C05072=1153.028,-21.073,-46.585,179.547,6.067,149.224
C05073=1153.033,-21.323,-46.572,179.545,6.067,149.225
C05074=1153.038,-21.572,-46.559,179.542,6.066,149.226
C05075=1153.044,-21.822,-46.547,179.540,6.065,149.226
C05076=1153.049,-22.071,-46.535,179.537,6.065,149.227
C05077=1153.054,-22.321,-46.523,179.535,6.064,149.227
C05078=1153.059,-22.571,-46.510,179.532,6.064,149.228
C05079=1153.064,-22.820,-46.498,179.530,6.063,149.228
C05080=1153.070,-23.070,-46.486,179.527,6.063,149.229
C05081=1153.075,-23.319,-46.473,179.525,6.062,149.230
C05082=1153.080,-23.569,-46.461,179.523,6.061,149.230
C05083=1153.085,-23.818,-46.449,179.520,6.060,149.231
C05084=1153.091,-24.089,-46.436,179.518,6.060,149.231
C05085=1153.097,-24.359,-46.422,179.516,6.059,149.232
C05086=1153.102,-24.628,-46.409,179.513,6.059,149.233
C05087=1153.108,-24.899,-46.396,179.510,6.058,149.233
C05088=1153.113,-25.148,-46.383,179.508,6.058,149.234
C05089=1153.118,-25.398,-46.371,179.505,6.057,149.235
C05090=1153.124,-25.648,-46.359,179.503,6.056,149.235
C05091=1153.129,-25.897,-46.347,179.501,6.056,149.236
C05092=1153.134,-26.147,-46.335,179.498,6.055,149.236
C05093=1153.139,-26.397,-46.322,179.496,6.055,149.237
C05094=1153.144,-26.646,-46.311,179.494,6.054,149.237
C05095=1153.149,-26.896,-46.298,179.491,6.054,149.238
C05096=1153.155,-27.145,-46.287,179.489,6.053,149.238
C05097=1153.160,-27.395,-46.274,179.487,6.052,149.239
C05098=1153.165,-27.645,-46.262,179.484,6.052,149.240
C05099=1153.171,-27.895,-46.250,179.482,6.051,149.240
C05100=1153.176,-28.144,-46.238,179.479,6.050,149.241
C05101=1153.180,-28.394,-46.226,179.477,6.050,149.241
C05102=1153.186,-28.644,-46.214,179.474,6.049,149.242
C05103=1153.191,-28.893,-46.202,179.472,6.048,149.242
C05104=1153.196,-29.143,-46.190,179.469,6.048,149.243
C05105=1153.202,-29.392,-46.177,179.467,6.047,149.244
C05106=1153.207,-29.642,-46.165,179.464,6.047,149.244
C05107=1153.212,-29.892,-46.154,179.462,6.046,149.245
C05108=1153.217,-30.141,-46.142,179.460,6.045,149.246
C05109=1153.222,-30.391,-46.130,179.457,6.045,149.246
C05110=1153.228,-30.641,-46.118,179.455,6.044,149.247
C05111=1153.232,-30.891,-46.106,179.453,6.044,149.247
C05112=1153.237,-31.140,-46.094,179.451,6.044,149.248
C05113=1153.243,-31.390,-46.082,179.448,6.043,149.248
C05114=1153.248,-31.640,-46.070,179.446,6.043,149.249
C05115=1153.253,-31.889,-46.058,179.444,6.042,149.249
C05116=1153.258,-32.139,-46.046,179.441,6.041,149.250
C05117=1153.264,-32.389,-46.034,179.439,6.041,149.251
C05118=1153.269,-32.639,-46.022,179.437,6.040,149.251
C05119=1153.274,-32.888,-46.010,179.434,6.039,149.252
C05120=1153.279,-33.137,-45.999,179.432,6.039,149.252
C05121=1153.284,-33.387,-45.987,179.429,6.038,149.253
C05122=1153.290,-33.637,-45.975,179.427,6.037,149.253
C05123=1153.295,-33.886,-45.964,179.424,6.037,149.254
C05124=1153.300,-34.136,-45.951,179.422,6.036,149.255
C05125=1153.305,-34.386,-45.939,179.419,6.036,149.255
C05126=1153.311,-34.635,-45.928,179.417,6.035,149.256
C05127=1153.316,-34.885,-45.916,179.414,6.035,149.257
C05128=1153.321,-35.135,-45.904,179.413,6.035,149.257
C05129=1153.326,-35.384,-45.892,179.410,6.034,149.258
C05130=1153.331,-35.634,-45.880,179.408,6.033,149.258
C05131=1153.336,-35.884,-45.869,179.405,6.033,149.259
C05132=1153.342,-36.134,-45.857,179.403,6.032,149.259
C05133=1153.347,-36.383,-45.846,179.401,6.031,149.260
C05134=1153.352,-36.633,-45.834,179.398,6.031,149.261
C05135=1153.358,-36.883,-45.822,179.396,6.030,149.261
C05136=1153.363,-37.132,-45.811,179.393,6.030,149.262
C05137=1153.368,-37.382,-45.798,179.391,6.029,149.262
C05138=1153.373,-37.632,-45.786,179.389,6.028,149.263
C05139=1153.378,-37.881,-45.775,179.386,6.028,149.263
C05140=1153.383,-38.131,-45.763,179.384,6.027,149.264
C05141=1153.389,-38.380,-45.752,179.382,6.027,149.265
C05142=1153.394,-38.630,-45.740,179.380,6.027,149.265
C05143=1153.399,-38.880,-45.728,179.377,6.026,149.266
C05144=1153.404,-39.129,-45.717,179.375,6.026,149.266
C05145=1153.410,-39.379,-45.705,179.372,6.025,149.267
C05146=1153.415,-39.629,-45.693,179.370,6.024,149.267
C05147=1153.420,-39.878,-45.682,179.368,6.024,149.268
C05148=1153.426,-40.128,-45.670,179.365,6.023,149.269
C05149=1153.430,-40.378,-45.659,179.363,6.022,149.269
C05150=1153.436,-40.628,-45.647,179.361,6.022,149.270
C05151=1153.440,-40.877,-45.636,179.358,6.021,149.270
C05152=1153.447,-41.127,-45.624,179.356,6.021,149.271
C05153=1153.452,-41.377,-45.613,179.354,6.021,149.272
C05154=1153.457,-41.626,-45.601,179.351,6.020,149.272
C05155=1153.462,-41.876,-45.589,179.349,6.020,149.273
C05156=1153.467,-42.126,-45.578,179.347,6.019,149.273
C05157=1153.473,-42.375,-45.567,179.344,6.018,149.274
C05158=1153.477,-42.625,-45.555,179.342,6.018,149.274
C05159=1153.483,-42.875,-45.543,179.340,6.017,149.275
C05160=1153.488,-43.124,-45.532,179.337,6.016,149.276
C05161=1153.493,-43.374,-45.520,179.335,6.016,149.276
C05162=1153.499,-43.624,-45.510,179.333,6.016,149.277
C05163=1153.504,-43.874,-45.498,179.331,6.015,149.277
C05164=1153.509,-44.123,-45.487,179.328,6.015,149.278
C05165=1153.514,-44.373,-45.475,179.326,6.014,149.278
C05166=1153.519,-44.622,-45.464,179.323,6.014,149.279
C05167=1153.525,-44.872,-45.452,179.321,6.013,149.280
C05168=1153.530,-45.122,-45.441,179.319,6.012,149.280
C05169=1153.535,-45.372,-45.429,179.317,6.012,149.281
C05170=1153.541,-45.621,-45.419,179.314,6.012,149.281
C05171=1153.546,-45.871,-45.407,179.312,6.011,149.282
C05172=1153.551,-46.121,-45.396,179.310,6.010,149.282
C05173=1153.555,-46.370,-45.384,179.307,6.010,149.283
C05174=1153.561,-46.620,-45.373,179.305,6.009,149.284
C05175=1153.566,-46.869,-45.362,179.302,6.009,149.284
C05176=1153.572,-47.120,-45.350,179.300,6.008,149.285
C05177=1153.577,-47.369,-45.339,179.298,6.008,149.285
C05178=1153.583,-47.619,-45.328,179.296,6.008,149.286
C05179=1153.587,-47.868,-45.316,179.293,6.007,149.286
C05180=1153.592,-48.118,-45.306,179.291,6.007,149.287
C05181=1153.598,-48.368,-45.294,179.289,6.006,149.288
C05182=1153.603,-48.617,-45.283,179.286,6.005,149.288
C05183=1153.608,-48.867,-45.271,179.284,6.005,149.289
C05184=1153.614,-49.117,-45.261,179.282,6.005,149.289
C05185=1153.619,-49.366,-45.249,179.279,6.004,149.290
C05186=1153.624,-49.616,-45.238,179.277,6.004,149.291
C05187=1153.629,-49.866,-45.226,179.275,6.003,149.291
C05188=1153.635,-50.136,-45.214,179.272,6.003,149.292
C05189=1153.641,-50.407,-45.202,179.270,6.002,149.292
C05190=1153.647,-50.678,-45.190,179.267,6.001,149.293
C05191=1153.652,-50.948,-45.179,179.264,6.001,149.294
C05192=1153.657,-51.198,-45.167,179.262,6.000,149.294
C05193=1153.663,-51.448,-45.157,179.260,5.999,149.295
C05194=1153.668,-51.697,-45.145,179.258,6.000,149.295
C05195=1153.673,-51.947,-45.133,179.256,5.999,149.296
C05196=1153.679,-52.197,-45.123,179.253,5.999,149.297
C05197=1153.683,-52.446,-45.112,179.251,5.998,149.297
C05198=1153.689,-52.696,-45.100,179.248,5.997,149.298
C05199=1153.694,-52.946,-45.090,179.246,5.997,149.298
C05200=1153.699,-53.196,-45.078,179.244,5.997,149.299
C05201=1153.705,-53.446,-45.067,179.242,5.996,149.299
C05202=1153.710,-53.695,-45.056,179.240,5.995,149.300
C05203=1153.715,-53.945,-45.045,179.237,5.995,149.301
C05204=1153.720,-54.194,-45.035,179.235,5.994,149.301
C05205=1153.726,-54.444,-45.023,179.232,5.994,149.302
C05206=1153.731,-54.694,-45.012,179.230,5.994,149.302
C05207=1153.736,-54.943,-45.002,179.228,5.993,149.303
C05208=1153.741,-55.194,-44.991,179.226,5.993,149.303
C05209=1153.747,-55.443,-44.979,179.223,5.992,149.304
C05210=1153.752,-55.692,-44.968,179.221,5.991,149.305
C05211=1153.757,-55.943,-44.958,179.219,5.991,149.305
C05212=1153.762,-56.192,-44.947,179.216,5.991,149.306
C05213=1153.768,-56.442,-44.935,179.214,5.990,149.306
C05214=1153.772,-56.692,-44.924,179.212,5.990,149.307
C05215=1153.778,-56.941,-44.914,179.209,5.989,149.307
C05216=1153.783,-57.191,-44.903,179.207,5.988,149.308
C05217=1153.788,-57.440,-44.892,179.205,5.989,149.309
C05218=1153.794,-57.690,-44.881,179.203,5.988,149.309
C05219=1153.799,-57.940,-44.870,179.200,5.988,149.310
C05220=1153.804,-58.190,-44.859,179.198,5.987,149.310
C05221=1153.809,-58.440,-44.848,179.196,5.986,149.311
C05222=1153.814,-58.689,-44.838,179.194,5.986,149.312
C05223=1153.819,-58.939,-44.827,179.192,5.986,149.312
C05224=1153.826,-59.189,-44.816,179.189,5.985,149.313
C05225=1153.830,-59.438,-44.805,179.187,5.984,149.313
C05226=1153.836,-59.688,-44.795,179.184,5.984,149.314
C05227=1153.841,-59.938,-44.783,179.183,5.984,149.314
C05228=1153.846,-60.187,-44.773,179.180,5.983,149.315
C05229=1153.851,-60.437,-44.763,179.178,5.983,149.316
C05230=1153.857,-60.686,-44.752,179.176,5.982,149.316
C05231=1153.862,-60.937,-44.741,179.173,5.982,149.317
C05232=1153.867,-61.187,-44.729,179.171,5.982,149.317
C05233=1153.873,-61.436,-44.719,179.169,5.981,149.318
C05234=1153.878,-61.686,-44.708,179.166,5.981,149.318
C05235=1153.883,-61.935,-44.698,179.164,5.980,149.319
C05236=1153.888,-62.185,-44.687,179.162,5.979,149.320
C05237=1153.893,-62.435,-44.677,179.160,5.979,149.320
C05238=1153.898,-62.685,-44.665,179.157,5.979,149.321
C05239=1153.904,-62.934,-44.655,179.155,5.978,149.321
C05240=1153.909,-63.184,-44.645,179.153,5.977,149.322
C05241=1153.915,-63.434,-44.633,179.150,5.977,149.322
C05242=1153.920,-63.684,-44.623,179.149,5.977,149.323
C05243=1153.925,-63.933,-44.612,179.146,5.977,149.324
C05244=1153.930,-64.183,-44.601,179.144,5.976,149.324
C05245=1153.936,-64.433,-44.591,179.142,5.975,149.325
C05246=1153.941,-64.682,-44.581,179.140,5.975,149.325
C05247=1153.946,-64.932,-44.570,179.137,5.975,149.326
C05248=1153.952,-65.181,-44.559,179.135,5.974,149.326
C05249=1153.957,-65.432,-44.549,179.132,5.974,149.327
C05250=1153.962,-65.681,-44.538,179.131,5.974,149.327
C05251=1153.967,-65.931,-44.528,179.128,5.973,149.328
C05252=1153.972,-66.180,-44.517,179.126,5.972,149.329
C05253=1153.977,-66.431,-44.506,179.123,5.972,149.329
C05254=1153.983,-66.680,-44.496,179.121,5.971,149.330
C05255=1153.988,-66.930,-44.486,179.120,5.971,149.330
C05256=1153.993,-67.179,-44.475,179.117,5.971,149.331
C05257=1153.999,-67.429,-44.464,179.115,5.970,149.331
C05258=1154.004,-67.679,-44.454,179.112,5.970,149.332
C05259=1154.009,-67.929,-44.444,179.110,5.970,149.333
C05260=1154.014,-68.179,-44.433,179.108,5.969,149.333
C05261=1154.020,-68.428,-44.423,179.106,5.968,149.334
C05262=1154.025,-68.678,-44.412,179.103,5.968,149.334
C05263=1154.030,-68.928,-44.401,179.101,5.968,149.335
C05264=1154.036,-69.177,-44.391,179.099,5.967,149.336
C05265=1154.041,-69.427,-44.381,179.097,5.967,149.336
C05266=1154.047,-69.677,-44.370,179.094,5.966,149.337
C05267=1154.052,-69.927,-44.360,179.093,5.966,149.337
C05268=1154.057,-70.177,-44.350,179.090,5.966,149.338
C05269=1154.062,-70.426,-44.339,179.088,5.965,149.338
C05270=1154.067,-70.676,-44.328,179.086,5.964,149.339
C05271=1154.072,-70.925,-44.318,179.084,5.965,149.340
C05272=1154.078,-71.175,-44.308,179.081,5.964,149.340
C05273=1154.083,-71.425,-44.298,179.079,5.963,149.341
C05274=1154.089,-71.674,-44.287,179.076,5.963,149.341
C05275=1154.094,-71.925,-44.277,179.075,5.963,149.342
C05276=1154.099,-72.174,-44.267,179.072,5.962,149.342
C05277=1154.105,-72.424,-44.256,179.070,5.962,149.343
C05278=1154.110,-72.674,-44.246,179.068,5.961,149.343
C05279=1154.115,-72.924,-44.236,179.066,5.961,149.344
C05280=1154.121,-73.173,-44.225,179.064,5.960,149.345
C05281=1154.125,-73.423,-44.215,179.061,5.960,149.345
C05282=1154.131,-73.673,-44.205,179.059,5.960,149.346
C05283=1154.136,-73.922,-44.195,179.057,5.959,149.346
C05284=1154.141,-74.172,-44.184,179.054,5.959,149.347
C05285=1154.147,-74.422,-44.174,179.052,5.958,149.347
C05286=1154.153,-74.671,-44.164,179.051,5.958,149.348
C05287=1154.158,-74.922,-44.154,179.048,5.958,149.349
C05288=1154.163,-75.171,-44.143,179.046,5.957,149.349
C05289=1154.168,-75.420,-44.134,179.043,5.957,149.350
C05290=1154.173,-75.671,-44.123,179.042,5.957,149.350
C05291=1154.179,-75.920,-44.113,179.039,5.956,149.351
C05292=1154.185,-76.192,-44.101,179.037,5.955,149.351
C05293=1154.190,-76.462,-44.091,179.034,5.955,149.352
C05294=1154.196,-76.734,-44.079,179.032,5.954,149.353
C05295=1154.201,-77.005,-44.068,179.030,5.955,149.353
C05296=1154.207,-77.255,-44.058,179.028,5.954,149.354
C05297=1154.213,-77.504,-44.048,179.025,5.953,149.354
C05298=1154.218,-77.754,-44.039,179.023,5.953,149.355
C05299=1154.223,-78.004,-44.028,179.021,5.953,149.356
C05300=1154.228,-78.254,-44.018,179.019,5.952,149.356
C05301=1154.234,-78.504,-44.008,179.016,5.952,149.357
C05302=1154.239,-78.754,-43.997,179.015,5.952,149.357
C05303=1154.244,-79.003,-43.988,179.012,5.951,149.358
C05304=1154.249,-79.253,-43.978,179.010,5.951,149.358
C05305=1154.255,-79.502,-43.967,179.008,5.951,149.359
C05306=1154.260,-79.753,-43.958,179.006,5.950,149.360
C05307=1154.265,-80.002,-43.948,179.003,5.949,149.360
C05308=1154.271,-80.252,-43.938,179.001,5.949,149.361
C05309=1154.276,-80.501,-43.928,178.999,5.949,149.361
C05310=1154.281,-80.751,-43.918,178.997,5.948,149.362
C05311=1154.286,-81.001,-43.907,178.995,5.947,149.362
C05312=1154.292,-81.251,-43.898,178.993,5.948,149.363
C05313=1154.298,-81.501,-43.888,178.990,5.947,149.363
C05314=1154.302,-81.750,-43.878,178.988,5.946,149.364
C05315=1154.308,-82.000,-43.867,178.986,5.947,149.365
C05316=1154.314,-82.250,-43.858,178.984,5.946,149.365
C05317=1154.318,-82.499,-43.848,178.981,5.946,149.366
C05318=1154.324,-82.749,-43.838,178.980,5.946,149.366
C05319=1154.329,-82.999,-43.828,178.977,5.945,149.367
C05320=1154.334,-83.248,-43.818,178.975,5.944,149.367
C05321=1154.340,-83.499,-43.808,178.973,5.944,149.368
C05322=1154.345,-83.748,-43.798,178.971,5.944,149.368
C05323=1154.350,-83.998,-43.788,178.968,5.943,149.369
C05324=1154.356,-84.248,-43.779,178.966,5.943,149.370
C05325=1154.361,-84.498,-43.769,178.965,5.943,149.370
C05326=1154.366,-84.747,-43.759,178.962,5.942,149.371
C05327=1154.372,-84.997,-43.749,178.960,5.941,149.371
C05328=1154.377,-85.247,-43.739,178.958,5.941,149.372
C05329=1154.382,-85.497,-43.729,178.955,5.941,149.373
C05330=1154.387,-85.746,-43.719,178.953,5.940,149.373
C05331=1154.392,-85.996,-43.710,178.952,5.940,149.373
C05332=1154.398,-86.246,-43.700,178.949,5.940,149.374
C05333=1154.404,-86.495,-43.690,178.947,5.939,149.375
C05334=1154.408,-86.746,-43.680,178.945,5.939,149.375
C05335=1154.414,-86.995,-43.670,178.943,5.939,149.376
C05336=1154.419,-87.244,-43.661,178.940,5.938,149.376
C05337=1154.425,-87.495,-43.651,178.939,5.938,149.377
C05338=1154.430,-87.744,-43.641,178.936,5.938,149.378
C05339=1154.435,-87.994,-43.632,178.934,5.937,149.378
C05340=1154.440,-88.244,-43.621,178.932,5.937,149.379
C05341=1154.445,-88.493,-43.612,178.930,5.937,149.379
C05342=1154.451,-88.744,-43.602,178.927,5.936,149.380
C05343=1154.456,-88.993,-43.593,178.926,5.936,149.380
C05344=1154.462,-89.243,-43.583,178.923,5.935,149.381
C05345=1154.467,-89.492,-43.574,178.921,5.935,149.381
C05346=1154.472,-89.742,-43.563,178.919,5.935,149.382
C05347=1154.478,-89.993,-43.554,178.917,5.934,149.383
C05348=1154.483,-90.242,-43.544,178.914,5.934,149.383
C05349=1154.488,-90.492,-43.534,178.913,5.934,149.384
C05350=1154.493,-90.741,-43.525,178.910,5.933,149.384
C05351=1154.499,-90.991,-43.515,178.909,5.933,149.385
C05352=1154.504,-91.241,-43.506,178.906,5.932,149.385
C05353=1154.510,-91.491,-43.496,178.904,5.932,149.386
C05354=1154.515,-91.740,-43.487,178.902,5.932,149.386
C05355=1154.521,-91.990,-43.477,178.900,5.931,149.387
C05356=1154.525,-92.240,-43.467,178.898,5.931,149.387
C05357=1154.531,-92.490,-43.458,178.896,5.931,149.388
C05358=1154.536,-92.740,-43.448,178.893,5.930,149.389
C05359=1154.542,-92.990,-43.439,178.891,5.929,149.389
C05360=1154.547,-93.239,-43.429,178.889,5.930,149.390
C05361=1154.552,-93.489,-43.419,178.887,5.929,149.390
C05362=1154.557,-93.738,-43.410,178.885,5.928,149.391
C05363=1154.563,-93.989,-43.400,178.883,5.929,149.391
C05364=1154.568,-94.238,-43.391,178.881,5.928,149.392
C05365=1154.573,-94.488,-43.382,178.879,5.928,149.392
C05366=1154.579,-94.737,-43.372,178.877,5.927,149.393
C05367=1154.584,-94.987,-43.363,178.874,5.927,149.394
C05368=1154.590,-95.237,-43.353,178.873,5.927,149.394
C05369=1154.595,-95.486,-43.344,178.870,5.926,149.395
C05370=1154.601,-95.737,-43.334,178.868,5.926,149.395
C05371=1154.606,-95.986,-43.325,178.866,5.926,149.396
C05372=1154.610,-96.236,-43.315,178.864,5.925,149.396
C05373=1154.616,-96.486,-43.305,178.862,5.925,149.397
C05374=1154.621,-96.736,-43.296,178.860,5.925,149.397
C05375=1154.627,-96.986,-43.287,178.857,5.924,149.398
C05376=1154.632,-97.235,-43.277,178.856,5.924,149.398
C05377=1154.638,-97.485,-43.268,178.853,5.924,149.399
C05378=1154.643,-97.735,-43.259,178.851,5.923,149.400
C05379=1154.648,-97.984,-43.249,178.849,5.923,149.400
C05380=1154.653,-98.235,-43.240,178.847,5.923,149.401
C05381=1154.659,-98.484,-43.231,178.845,5.923,149.401
C05382=1154.663,-98.734,-43.221,178.843,5.922,149.402
C05383=1154.669,-98.984,-43.212,178.841,5.921,149.402
C05384=1154.675,-99.234,-43.203,178.839,5.921,149.403
C05385=1154.680,-99.483,-43.192,178.836,5.921,149.403
C05386=1154.685,-99.733,-43.184,178.835,5.921,149.404
C05387=1154.690,-99.983,-43.175,178.832,5.920,149.405
C05388=1154.696,-100.232,-43.164,178.830,5.920,149.405
C05389=1154.701,-100.482,-43.156,178.828,5.920,149.406
C05390=1154.706,-100.732,-43.147,178.826,5.919,149.406
C05391=1154.712,-100.982,-43.137,178.824,5.919,149.407
C05392=1154.717,-101.232,-43.128,178.822,5.918,149.407
C05393=1154.722,-101.481,-43.119,178.820,5.918,149.408
C05394=1154.728,-101.732,-43.109,178.818,5.918,149.408
C05395=1154.733,-101.981,-43.100,178.815,5.917,149.409
C05396=1154.740,-102.253,-43.090,178.813,5.917,149.410
C05397=1154.745,-102.525,-43.080,178.811,5.917,149.410
C05398=1154.750,-102.796,-43.070,178.809,5.916,149.411
C05399=1154.756,-103.069,-43.060,178.806,5.916,149.411
C05400=1154.762,-103.319,-43.051,178.805,5.916,149.412
C05401=1154.767,-103.568,-43.041,178.802,5.915,149.412
C05402=1154.772,-103.818,-43.032,178.800,5.914,149.413
C05403=1154.778,-104.068,-43.023,178.798,5.915,149.414
C05404=1154.783,-104.318,-43.014,178.796,5.914,149.414
C05405=1154.789,-104.567,-43.005,178.794,5.914,149.415
C05406=1154.794,-104.817,-42.996,178.792,5.913,149.415
C05407=1154.799,-105.066,-42.987,178.790,5.913,149.416
C05408=1154.805,-105.317,-42.977,178.788,5.913,149.416
C05409=1154.810,-105.566,-42.969,178.786,5.912,149.417
C05410=1154.815,-105.816,-42.960,178.784,5.912,149.417
C05411=1154.820,-106.066,-42.951,178.781,5.912,149.418
C05412=1154.826,-106.316,-42.941,178.780,5.912,149.418
C05413=1154.831,-106.566,-42.932,178.778,5.911,149.419
C05414=1154.836,-106.815,-42.923,178.775,5.910,149.419
C05415=1154.842,-107.065,-42.914,178.773,5.911,149.420
C05416=1154.847,-107.315,-42.905,178.771,5.910,149.421
C05417=1154.853,-107.565,-42.896,178.770,5.910,149.421
C05418=1154.858,-107.814,-42.887,178.767,5.909,149.422
C05419=1154.864,-108.064,-42.878,178.765,5.910,149.422
C05420=1154.869,-108.314,-42.869,178.763,5.909,149.423
C05421=1154.874,-108.564,-42.860,178.761,5.908,149.423
C05422=1154.880,-108.814,-42.851,178.759,5.908,149.424
C05423=1154.885,-109.064,-42.842,178.757,5.908,149.424
C05424=1154.890,-109.313,-42.832,178.755,5.908,149.425
C05425=1154.896,-109.562,-42.824,178.753,5.907,149.425
C05426=1154.901,-109.812,-42.815,178.751,5.907,149.426
C05427=1154.906,-110.062,-42.806,178.749,5.907,149.427
C05428=1154.912,-110.312,-42.796,178.746,5.906,149.427
C05429=1154.917,-110.562,-42.788,178.745,5.906,149.428
C05430=1154.922,-110.812,-42.779,178.743,5.905,149.428
C05431=1154.927,-111.062,-42.770,178.741,5.905,149.429
C05432=1154.933,-111.311,-42.761,178.738,5.905,149.429
C05433=1154.938,-111.561,-42.752,178.737,5.905,149.430
C05434=1154.943,-111.811,-42.743,178.735,5.904,149.430
C05435=1154.949,-112.061,-42.734,178.732,5.904,149.431
C05436=1154.955,-112.311,-42.725,178.730,5.904,149.431
C05437=1154.960,-112.561,-42.716,178.728,5.903,149.432
C05438=1154.965,-112.810,-42.708,178.726,5.903,149.432
C05439=1154.971,-113.060,-42.699,178.724,5.903,149.433
C05440=1154.976,-113.310,-42.691,178.723,5.903,149.433
C05441=1154.981,-113.560,-42.682,178.720,5.902,149.434
C05442=1154.986,-113.810,-42.673,178.718,5.902,149.435
C05443=1154.992,-114.060,-42.664,178.716,5.902,149.435
C05444=1154.997,-114.309,-42.655,178.715,5.902,149.436
C05445=1155.003,-114.559,-42.646,178.712,5.901,149.436
C05446=1155.008,-114.809,-42.637,178.710,5.900,149.437
C05447=1155.014,-115.059,-42.628,178.708,5.900,149.437
C05448=1155.019,-115.308,-42.619,178.706,5.900,149.438
C05449=1155.025,-115.558,-42.611,178.704,5.900,149.438
C05450=1155.030,-115.807,-42.602,178.702,5.899,149.439
C05451=1155.035,-116.058,-42.593,178.700,5.899,149.439
C05452=1155.040,-116.308,-42.585,178.698,5.899,149.440
C05453=1155.046,-116.557,-42.576,178.696,5.899,149.440
C05454=1155.051,-116.807,-42.567,178.694,5.898,149.441
C05455=1155.056,-117.057,-42.558,178.692,5.898,149.441
C05456=1155.062,-117.306,-42.549,178.690,5.898,149.442
C05457=1155.067,-117.556,-42.540,178.688,5.898,149.443
C05458=1155.073,-117.806,-42.533,178.686,5.897,149.443
C05459=1155.078,-118.056,-42.524,178.684,5.896,149.444
C05460=1155.083,-118.306,-42.515,178.682,5.896,149.444
C05461=1155.088,-118.556,-42.506,178.680,5.896,149.445
C05462=1155.094,-118.805,-42.497,178.678,5.896,149.445
C05463=1155.099,-119.055,-42.489,178.676,5.895,149.446
C05464=1155.105,-119.305,-42.480,178.674,5.895,149.446
C05465=1155.110,-119.555,-42.471,178.672,5.894,149.447
C05466=1155.116,-119.804,-42.463,178.670,5.895,149.447
C05467=1155.121,-120.054,-42.454,178.668,5.894,149.448
C05468=1155.126,-120.304,-42.446,178.666,5.894,149.448
C05469=1155.132,-120.554,-42.437,178.664,5.893,149.449
C05470=1155.137,-120.803,-42.428,178.662,5.893,149.449
C05471=1155.142,-121.053,-42.420,178.660,5.893,149.450
C05472=1155.148,-121.303,-42.411,178.658,5.893,149.451
C05473=1155.154,-121.553,-42.403,178.656,5.892,149.451
C05474=1155.159,-121.803,-42.394,178.654,5.892,149.452
C05475=1155.163,-122.052,-42.386,178.652,5.892,149.452
C05476=1155.169,-122.303,-42.377,178.650,5.892,149.453
C05477=1155.174,-122.552,-42.369,178.648,5.891,149.453
C05478=1155.180,-122.802,-42.360,178.646,5.891,149.454
C05479=1155.185,-123.052,-42.351,178.644,5.891,149.454
C05480=1155.191,-123.301,-42.343,178.642,5.890,149.455
C05481=1155.196,-123.551,-42.334,178.640,5.890,149.455
C05482=1155.201,-123.801,-42.325,178.638,5.889,149.456
C05483=1155.207,-124.051,-42.318,178.636,5.889,149.456
C05484=1155.212,-124.301,-42.309,178.634,5.889,149.457
C05485=1155.218,-124.551,-42.300,178.632,5.889,149.457
C05486=1155.223,-124.800,-42.293,178.630,5.888,149.458
C05487=1155.228,-125.050,-42.284,178.628,5.888,149.458
C05488=1155.233,-125.300,-42.275,178.626,5.887,149.459
C05489=1155.239,-125.549,-42.267,178.625,5.887,149.459
C05490=1155.245,-125.799,-42.258,178.622,5.887,149.460
C05491=1155.250,-126.049,-42.249,178.620,5.887,149.461
C05492=1155.256,-126.299,-42.241,178.618,5.886,149.461
C05493=1155.260,-126.548,-42.233,178.616,5.886,149.461
C05494=1155.266,-126.799,-42.225,178.614,5.886,149.462
C05495=1155.271,-127.048,-42.216,178.613,5.886,149.462
C05496=1155.277,-127.298,-42.208,178.610,5.885,149.463
